(* CODESYS project 117_1_V0.5.project

Project tree, tasks and I/O mapping:
  Device : XSLH-30A32, Wuxi Xinje Electric Co.,Ltd., version 3.5.15.40_2.2.0_2023.07.04
      unmapped channels: IN, OUT
    application Application
      libraries: Standard, * (System); Util, * (System); CmpIecTask, 3.5.21.0 (System); Time and Date, 3.5.17.0 (3S - Smart Software Solutions GmbH); Asynchronous Job  Manager, 3.5.19.0 (3S - Smart Software Solutions GmbH); CmpEventMgr, 3.5.14.0 (System); Component Manager, 3.5.13.0 (System); CmpApp, 3.5.15.0 (System)
      task EtherCAT_Task (cyclic, interval 4 ms, priority 1) calls nothing
      task MainTask (cyclic, interval 4 ms, priority 8) calls MAIN
      6.Logic/
        data type STATUS
        function block StandLogic [ST]: _move_algorythm, _get_status, _change_control_mode, _jogging, _init, _alarm_notification, _read_inputs, _collect_errors, _driver_power, _write_outputs, _reset_alarms, _check_exciter, read_control_mode, _check_removing_limit_switch
        data type AUTO_MOVE_STEPS
        data type CONTROL_MODE
      Symbols
      0.TaskData/
        TimeManager_Structs/
          data type MEASUREMENT_UNITS
          data type TYPE_
        function block TimeManager [ST]: get_date_time, get_interval_time_type_INT, get_interval_time_type_REAL, get_interval_time_type_TIME, get_interval_time_type_UINT, get_cycle_count
      1.IO/
        Output/
          function block OutputManager [ST]: set_data
          data type DQ_VARS
        Input/
          function block InputManager [ST]: get_analog_data, get_discrete_data
          data type ALL_DI
          data type ALL_AI
      2.PID/
        PID_Structs/
          data type PID_STATUS_UDT
          data type PID_DIRECTION_UDT
          data type PID_DIAGNOSTIC_UDT
          data type PID_PARAMETERS_UDT
        function block BasicPIDController [ST]: Set_Configuration, Get_Diagnostics, xDifferential, Enable, Disable, xSp, xError, xPv, xIntegral, xOutput, Reset, xProportional
      2.Exciter/
        SwitchingAndFeedbackControl/
          data type SW_STATUS
          function block SwitchingWithFeedbackControl [ST]
          function block WaitingTimer [ST]
      4.Servo/
        Servo_Structs/
          data type ERROR_INDEX
          data type SMC_ERROR_TO_STRING
        function block SM3ServoDriver [ST]: _error_handler, set_power_on, stop_follow_velocity, start_forward_jogging, get_power_status, set_power_off, stop_jogging, reset_errors, start_follow_velocity, get_axis_errors, start_backward_jogging, get_axis_communication
      5.PRG/
        program MAIN [ST]
    Modbus_TCP : Modbus TCP, Wuxi Xinje Electric Co.,Ltd., version 3.0.0.0
    SoftMotion General Axis Pool
    EtherCAT_Master_SoftMotion : EtherCAT Master SoftMotion, CODESYS, version 4.10.0.0
        settings: SlaveAutoRestart = True; NetworkName = 'eth1'; NetworkName = "eth1"; SrcAddress1 = 26855; SrcAddress2 = 1253576340; EnableSecondAdapter = False
      ECAT_2057P_16DO : ECAT-2057P(RevC.) 16 K. Dig. Aus. Source 40V 0.3A, ICP DAS Co., Ltd., order no. ECAT-2057P 16DO, version Revision=16#00400001
          settings: Physical Address of the Slave = 1002; AutoIncr Address of the Slave = 4294967295; StationAlias = 0; FMMU.Global Start Address = 16#02000000; FMMU.Physical Start Address = 16#0F00; FMMU.Access = 16#02; DC sync0 cycletime = 4000; DC sync1 cycletime = 4000
          unmapped channels: Output 0 to 7, Output 0 to 7, Output 0 to 7, Output 0 to 7, Output 0 to 7, Output 0 to 7, Output 0 to 7, Output 0 to 7, Output 8 to 15, Output 8 to 15, Output 8 to 15, Output 8 to 15, Output 8 to 15, Output 8 to 15, Output 8 to 15, Output 8 to 15
      SD700_ECAT_Drive : SD700_ECAT_V1.5_G, Shenzhen Veichi Electric Co., Ltd, order no. SD700_ECAT Drive, version Revision=16#02040608
          settings: Number of Inputs = 7; Number of Infos about Inputs = 7; EnableExpertSettings = True; Watchdog_Reg_0400 = 2498; Watchdog_Reg_0410 = 1000; Watchdog_Reg_0420 = 1000; Physical Address of the Slave = 1003; AutoIncr Address of the Slave = 4294967294; StationAlias = 0; Sync.Length = 18; FMMU.Global Start Address = 16#02000002; FMMU.Physical Start Address = 16#1100; FMMU.Access = 16#02; FMMU.Global Start Address = 16#01000002; FMMU.Length = 18; FMMU.Physical Start Address = 16#1400; FMMU.Access = 16#01; FMMU.Global Start Address = 16#00080000; FMMU.Physical Start Address = 16#080D; FMMU.Access = 16#01; DC sync0 cycletime = 4000; DC enable = 1; DC sync0 enable = 1; DC sync0 shift time = 0; DC sync1 cycletime = 4000; DC sync1 enable = 0; DC sync1 factor = 'x 1'; DC sync1 shift time = 0; Number of SDO = 3; Interpolation time period.Value = 4; RxTxPdo.NumberofEntries = 7; RxTxPdo.Index = 16#1A01; RxTxPdo.DependOnSlot = False; RxTxPdo.DependOnSlotGroup = False; RxTxPdo.OverwrittenByModule = False; Exclude = [16#1A00,16#1A02,16#1A03]; Status Word.Offset = 0; Status Word.DependOnSlot = False; Status Word.DependOnSlotGroup = False; ActualPosition.Offset = 0;
            ActualPosition.DependOnSlot = False; ActualPosition.DependOnSlotGroup = False; Velocity actual value.Offset = 0; Velocity actual value.DependOnSlot = False; Velocity actual value.DependOnSlotGroup = False; Un000.Index = 16#3000; Un000.SubIndex = 0; Un000.Size = 16; Un000.Offset = 0; Un000.DependOnSlot = False; Un000.DependOnSlotGroup = False; Un001.Index = 16#3001; Un001.SubIndex = 0; Un001.Size = 16; Un001.Offset = 0; Un001.DependOnSlot = False; Un001.DependOnSlotGroup = False; Un004.Index = 16#3004; Un004.SubIndex = 0; Un004.Size = 16; Un004.Offset = 0; Un004.DependOnSlot = False; Un004.DependOnSlotGroup = False; Un005.Index = 16#3005; Un005.SubIndex = 0; Un005.Size = 16; Un005.Offset = 0; Un005.DependOnSlot = False; Un005.DependOnSlotGroup = False; Status Word.Default = ''; Status Word.Comment = ''; ActualPosition.Default = ''; ActualPosition.Comment = ''; Velocity actual value.Default = ''; Velocity actual value.Comment = ''; Un000.Name = 'Un000'; Un000.DataType = 'INT'; Un000.Default = ''; Un000.Comment = ''; Un001.Name = 'Un001';
            Un001.DataType = 'INT'; Un001.Default = ''; Un001.Comment = ''; Un004.Name = 'Un004'; Un004.DataType = 'UINT'; Un004.Default = ''; Un004.Comment = ''; Un005.Name = 'Un005'; Un005.DataType = 'UINT'; Un005.Default = ''; Un005.Comment = ''
          unmapped channels: Control Word, TargetPosition, TargetVelocity, Status Word, ActualPosition, Velocity actual value, Un000, Un001, Un004, Un005
        SM_Drive_GenericDSP402 : SM_Drive_GenericDSP402, CODESYS, order no. 0, version 4.19.0.0
            settings: wDriveID = 0; dwRatioTechUnitsDenom = 83886080; eRampType = 0; ScalingIncs = 8388608; ScalingMotorTurns2 = 50; ScalingUnits = 5; AdrOffset_8010 = 4; BitOffset_8010 = 0; BitLength_8010 = 16; Address_8010 = '%QW2'; Type_8010 = 'UINT'; AddressPointer_8010 = ADR(%QW2); AdrOffset_8020 = 8; BitOffset_8020 = 0; BitLength_8020 = 32; Address_8020 = '%QD2'; Type_8020 = 'DINT'; AddressPointer_8020 = ADR(%QD2); AdrOffset_8030 = 12; BitOffset_8030 = 0; BitLength_8030 = 32; Address_8030 = '%QD3'; Type_8030 = 'DINT'; AddressPointer_8030 = ADR(%QD3); AdrOffset_8040 = 4294967295; BitOffset_8040 = 0; BitLength_8040 = 16; Address_8040 = ''; Type_8040 = 'INT'; AddressPointer_8040 = 0; AdrOffset_8050 = 4294967295; BitOffset_8050 = 0; BitLength_8050 = 8; Address_8050 = ''; Type_8050 = 'SINT'; AddressPointer_8050 = 0; AdrOffset_8060 = 4294967295; BitOffset_8060 = 0; BitLength_8060 = 16; Address_8060 = '';
              Type_8060 = 'UINT'; AddressPointer_8060 = 0; AdrOffset_8070 = 4294967295; BitOffset_8070 = 0; BitLength_8070 = 0; Address_8070 = ''; Type_8070 = ''; AddressPointer_8070 = 0; AdrOffset_8080 = 4294967295; BitOffset_8080 = 0; BitLength_8080 = 0; Address_8080 = ''; Type_8080 = ''; AddressPointer_8080 = 0; AdrOffset_8090 = 4294967295; BitOffset_8090 = 0; BitLength_8090 = 0; Address_8090 = ''; Type_8090 = ''; AddressPointer_8090 = 0; AdrOffset_8510 = 4; BitOffset_8510 = 0; BitLength_8510 = 16; Address_8510 = '%IW2'; Type_8510 = 'UINT'; AddressPointer_8510 = ADR(%IW2); AdrOffset_8520 = 8; BitOffset_8520 = 0; BitLength_8520 = 32; Address_8520 = '%ID2'; Type_8520 = 'DINT'; AddressPointer_8520 = ADR(%ID2); AdrOffset_8530 = 12; BitOffset_8530 = 0; BitLength_8530 = 32; Address_8530 = '%ID3'; Type_8530 = 'DINT'; AddressPointer_8530 = ADR(%ID3); AdrOffset_8540 = 4294967295; BitOffset_8540 = 0;
              BitLength_8540 = 16; Address_8540 = ''; Type_8540 = 'INT'; AddressPointer_8540 = 0; AdrOffset_8550 = 4294967295; BitOffset_8550 = 0; BitLength_8550 = 0; Address_8550 = ''; Type_8550 = ''; AddressPointer_8550 = 0; AdrOffset_8560 = 4294967295; BitOffset_8560 = 0; BitLength_8560 = 32; Address_8560 = ''; Type_8560 = 'UDINT'; AddressPointer_8560 = 0; AdrOffset_8570 = 4294967295; BitOffset_8570 = 0; BitLength_8570 = 16; Address_8570 = ''; Type_8570 = 'UINT'; AddressPointer_8570 = 0; AdrOffset_8580 = 4294967295; BitOffset_8580 = 0; BitLength_8580 = 32; Address_8580 = ''; Type_8580 = 'DINT'; AddressPointer_8580 = 0; AdrOffset_8590 = 4294967295; BitOffset_8590 = 0; BitLength_8590 = 0; Address_8590 = ''; Type_8590 = ''; AddressPointer_8590 = 0; AdrOffset_8600 = 4294967295; BitOffset_8600 = 0; BitLength_8600 = 0; Address_8600 = ''; Type_8600 = ''; AddressPointer_8600 = 0;
              AdrOffset_8600 = 4294967295; BitOffset_8600 = 0; BitLength_8600 = 0; Address_8610 = ''; Type_8610 = ''; AddressPointer_8610 = 0; AdrOffset_8620 = 4294967295; BitOffset_8620 = 0; BitLength_8620 = 0; Address_8620 = ''; Type_8620 = ''; AddressPointer_8620 = 0
      ECAT_2016N_1 : ECAT-2016N 1 K. Ana. Eingang, Diff., 16-bit, ICP DAS Co.LTD, order no. ECAT-2016N , version Revision=16#00100001
          settings: EnableExpertSettings = True; StationAlias = 0; DC sync0 cycletime = 4000; DC sync1 cycletime = 4000
          unmapped channels: Status__Underrange, Status__Overrange, Status__Limit 1, Status__Limit 1, Status__Limit 2, Status__Limit 2, Status__Error, ---, ---, ---, ---, ---, ---, ---, Status__TxPDO State, Status__TxPDO Toggle, Value
      ECAT_2053_16DI : ECAT-2053 16 K. Dig. Ein. Wet 50V, ICP DAS Co., Ltd., order no. ECAT-2053 16DI, version Revision=16#00000001
          settings: Physical Address of the Slave = 1001; StationAlias = 1001; Optional = False; DeviceIdenticationADO = 0; DeviceIdenticationMode = 0; FMMU.Global Start Address = 16#01000000; FMMU.Physical Start Address = 16#1000; FMMU.Access = 16#01; DC sync0 cycletime = 4000; DC sync1 cycletime = 4000
          unmapped channels: Input 0 to 7, Input 0 to 7, Input 0 to 7, Input 0 to 7, Input 0 to 7, Input 0 to 7, Input 0 to 7, Input 0 to 7, Input 8 to 15, Input 8 to 15, Input 8 to 15, Input 8 to 15, Input 8 to 15, Input 8 to 15, Input 8 to 15, Input 8 to 15
      ECAT_2016N : ECAT-2016N 1 K. Ana. Eingang, Diff., 16-bit, ICP DAS Co.LTD, order no. ECAT-2016N , version Revision=16#00100001
          settings: EnableExpertSettings = True; Physical Address of the Slave = 1004; AutoIncr Address of the Slave = 4294967293; StationAlias = 0; FMMU.Global Start Address = 16#0200000C; FMMU.Physical Start Address = 16#1100; FMMU.Access = 16#02; FMMU.Global Start Address = 16#01000014; FMMU.Physical Start Address = 16#1400; FMMU.Access = 16#01; FMMU.Global Start Address = 16#00080000; FMMU.StartBit = 1; FMMU.EndBit = 1; FMMU.Physical Start Address = 16#080D; FMMU.Access = 16#01; DC sync0 cycletime = 4000; DC enable = 0; DC sync0 enable = 0; DC sync0 shift time = 0; DC sync1 cycletime = 4000; DC sync1 enable = 0; DC sync1 shift time = 0; Number of SDO = 0
          unmapped channels: Status__Underrange, Status__Overrange, Status__Limit 1, Status__Limit 1, Status__Limit 2, Status__Limit 2, Status__Error, ---, ---, ---, ---, ---, ---, ---, Status__TxPDO State, Status__TxPDO Toggle, Value
      TEC_Sensor : TEC Sensor E101 mit 1 Magnet, ZDJY TEC Corp, order no. TEC Sensor, version Revision=16#000100C9
          settings: EnableExpertSettings = True; Physical Address of the Slave = 1005; AutoIncr Address of the Slave = 4294967292; StationAlias = 0; FMMU.Global Start Address = 16#01000018; FMMU.Physical Start Address = 16#1400; FMMU.Access = 16#01; DC sync0 cycletime = 4000; DC sync1 cycletime = 4000
          unmapped channels: Status 1, Position 1, Velocity 1
    Local High Speed IO
        unmapped channels: IN, OUT
  ГОСТ/
    data type E_I_II
    Р ИСО 15032-2001/
      data type E_A
      function block TestingForces_150321 [ST]
     Р53868-2021/
      data type E_P1_2
      function block TestingForces_53868 [ST]
    Р ИСО 10328-2021/
      function block TestingForces_10328 [ST]
      data type E_P3_8
*)

// Device/Application/4.Servo/Servo_Structs/ERROR_INDEX
TYPE ERROR_INDEX :
(
	communication,
	power,
	jogging,
	follow,
	reset,
	lastIndex
)UINT;
END_TYPE

// Device/Application/6.Logic/STATUS
{attribute 'strict'}
TYPE STATUS :
(
	NOT_COMMUNICATION,
	OFF,
	READY,
	MOVING,
	ERROR
);
END_TYPE

// ГОСТ/E_I_II
{attribute 'strict'}
TYPE E_I_II :
(
	I := 0,
	II := 1
);
END_TYPE

// Device/Application/2.Exciter/SwitchingAndFeedbackControl/SW_STATUS
{attribute 'qualified_only'}
{attribute 'strict'}
TYPE SW_STATUS :
(	
	NONE,
	WAITING,
	DONE,
	TIMEOUT_ERROR
);
END_TYPE

// ГОСТ/ Р53868-2021/E_P1_2
{attribute 'strict'}
TYPE E_P1_2 :
(
	P1:= 0,
	P2:= 1
);
END_TYPE

// ГОСТ/Р ИСО 15032-2001/E_A
{attribute 'strict'}
TYPE E_A :
(
	A60		:= 0,
	A80		:= 1,
	A100	:= 2
);
END_TYPE

// Device/Application/6.Logic/AUTO_MOVE_STEPS
{attribute 'strict'}
TYPE AUTO_MOVE_STEPS :
(
	AWAIT,
	INJECTION,
	RETENTION,
	FAILING
);
END_TYPE

// Device/Application/0.TaskData/TimeManager_Structs/MEASUREMENT_UNITS
{attribute 'strict'}
TYPE MEASUREMENT_UNITS  :
(
	MS,
	US
);
END_TYPE

// Device/Application/2.PID/PID_Structs/PID_STATUS_UDT
{attribute 'strict' := ''}
TYPE PID_STATUS_UDT :
(
	Disabled,
	Enabled
);
END_TYPE

// Device/Application/1.IO/Input/ALL_DI
{attribute 'strict'}
TYPE ALL_DI :
(
	inLiveCircuitsDC		,			
	inFirstAlarmMushroom	,
	inSecondAlarmMushroom	,
	inLiveCircuitsAC		,		
	inUpsDC_OK				,			
	inUpsBattaryBad			,		
	inUpsBattaryWork		,	
	inUpperLimitSwitch		,	
	inLowerLimitSwitch		,	
	inRemovingLimitSwitch	,
	inExciter				,		
	inBit11					,				
	inBit12					,				
	inLeftDoor				,			
	inRightDoor				,			
	inBit15					
);
END_TYPE

// Device/Application/2.PID/PID_Structs/PID_DIRECTION_UDT
{attribute 'strict' := ''}
TYPE PID_DIRECTION_UDT :
(
	///[0] Прямая работа: ошибка = SP - PV
	DIRECT,
	///[1] Обратная работа: ошибка = PV - SP
	REVERSE
);
END_TYPE

// Device/Application/6.Logic/CONTROL_MODE
{attribute 'strict'}
TYPE CONTROL_MODE :
(
	MANUAL	:= 10,
	AUTO	:= 20
);
END_TYPE

// Device/Application/2.PID/PID_Structs/PID_DIAGNOSTIC_UDT
TYPE PID_DIAGNOSTIC_UDT :
STRUCT
	Error			: REAL;
	PreviousError	: REAL;
	Proportional	: REAL;
	Integral		: REAL;
	Differential	: REAL;
	Status			: PID_STATUS_UDT;
	Direction		: PID_DIRECTION_UDT;
	Kp				: REAL;
	Ki				: REAL;
	Kd				: REAL;
	Ts				: TIME;
	MinOut			: REAL;
	MaxOut			: REAL;
END_STRUCT
END_TYPE

// ГОСТ/Р ИСО 10328-2021/E_P3_8
{attribute 'strict'}
TYPE E_P3_8 :
(
	P3:= 0,
	P4:= 1,
	P5:= 2,
	P6:= 3,
	P7:= 4,
	P8:= 5
	
);
END_TYPE

// Device/Application/2.PID/PID_Structs/PID_PARAMETERS_UDT
TYPE PID_PARAMETERS_UDT :
STRUCT
	Pv: REAL;
	Sp: REAL;
	Kp: REAL;
	Ki: REAL;
	Kd: REAL;
	Ts: TIME;
	MinOut: REAL;
	MaxOut: REAL;
	Direction: PID_DIRECTION_UDT;
END_STRUCT
END_TYPE

// Device/Application/1.IO/Input/ALL_AI
TYPE ALL_AI :
(
	tenza1000kgSensor,
	tenza50kgSensor	,
	motionSensor	,
    lastAnalogInIndex	
);
END_TYPE

// Device/Application/4.Servo/Servo_Structs/SMC_ERROR_TO_STRING
{attribute 'to_string'}
TYPE SMC_ERROR_TO_STRING :
(
	SMC_NO_ERROR := 0,
	SMC_DI_GENERAL_COMMUNICATION_ERROR := 1,
	SMC_DI_AXIS_ERROR := 2,
	SMC_DI_FIELDBUS_LOST_SYNCRONICITY := 3,
	SMC_DI_SWLIMITS_EXCEEDED := 10,
	SMC_DI_HWLIMITS_EXCEEDED := 11,
	SMC_DI_LINEAR_AXIS_OUTOFRANGE := 12,
	SMC_DI_HALT_OR_QUICKSTOP_NOT_SUPPORTED := 13,
	SMC_DI_VOLTAGE_DISABLED := 14,
	SMC_DI_IRREGULAR_ACTPOSITION := 15,
	SMC_DI_POSITIONLAGERROR := 16,
	SMC_DI_HOMING_ERROR := 17,
	SMC_DI_LICENSING_ERROR := 18,
	SMC_DI_DRIVE_LIMIT_ACTIVE := 19,
	SMC_REGULATOR_OR_START_NOT_SET := 20,
	SMC_WRONG_CONTROLLER_MODE := 21,
	SMC_INVALID_ACTION_FOR_LOGICAL := 25,
	SMC_AXIS_IS_NOT_OPERATIONAL := 27,
	SMC_AXIS_NOT_FOLLOWING_SETVALUES := 28,
	SMC_FB_WASNT_CALLED_DURING_MOTION := 30,
	SMC_AXIS_IS_NO_AXIS_REF := 31,
	SMC_AXIS_REF_CHANGED_DURING_OPERATION := 32,
	SMC_FB_ACTIVE_AXIS_DISABLED := 33,
	SMC_AXIS_NOT_READY_FOR_MOTION := 34,
	SMC_AXIS_ERROR_DURING_MOTION := 35,
	SMC_FB_CALLED_FROM_WRONG_TASK := 36,
	SMC_INVALID_DISTRIBUTED_CLOCKS_SETTINGS := 37,
	SMC_INVALID_TIMESTAMP := 38,
	SMC_AXIS_ERROR_DUE_TO_FB_ERROR := 39,
	SMC_VD_MAX_VELOCITY_EXCEEDED := 40,
	SMC_VD_MAX_ACCELERATION_EXCEEDED := 41,
	SMC_VD_MAX_DECELERATION_EXCEEDED := 42,
	SMC_3SH_INVALID_VELACC_VALUES := 50,
	SMC_3SH_MODE_NEEDS_HWLIMIT := 51,
	SMC_FRC_NO_FREE_HANDLE := 60,
	SMC_MAC_INITIALIZATION_FAILED := 65,
	SMC_MAC_INVALID_TASK_HANDLE := 66,
	SMC_MAC_TOO_MANY_TASKS := 67,
	SMC_MAC_ATOMIC_ADD_FAILED := 68,
	SMC_SDO_INVALID_DATALENGTH := 69,
	SMC_SCM_NOT_SUPPORTED := 70,
	SMC_SCM_AXIS_IN_WRONG_STATE := 71,
	SMC_SCM_INTERRUPTED := 72,
	SMC_ST_WRONG_CONTROLLER_MODE := 75,
	SMC_RAG_ERROR_DURING_STARTUP := 80,
	SMC_RAG_ERROR_AXIS_NOT_INITIALIZED := 81,
	SMC_PP_WRONG_AXIS_TYPE := 85,
	SMC_PP_NUMBER_OF_ABSOLUTE_BITS_INVALID := 86,
	SMC_NEGATIVE_MODULO_PERIOD := 87,
	SMC_CGR_ZERO_VALUES := 90,
	SMC_CGR_DRIVE_POWERED := 91,
	SMC_CGR_INVALID_POSPERIOD := 92,
	SMC_CGR_POSPERIOD_NOT_INTEGRAL := 93,
	SMC_FRACTION_TECH_UNITS_INVALID := 94,
	SMC_SCALING_PARAMETERS_NOT_POSITIVE := 95,
	SMC_SCALING_SETTINGS_TOO_LARGE := 96,
	SMC_MODULO_PERIOD_TOO_MANY_DIGITS := 97,
	SMC_P_FTASKCYCLE_EMPTY := 110,
	SMC_R_NO_ERROR_TO_RESET := 120,
	SMC_R_DRIVE_DOESNT_ANSWER := 121,
	SMC_R_ERROR_NOT_RESETTABLE := 122,
	SMC_R_DRIVE_DOESNT_ANSWER_IN_TIME := 123,
	SMC_R_CANNOT_RESET_COMMUNICATION_ERROR := 124,
	SMC_RP_PARAM_UNKNOWN := 130,
	SMC_RP_REQUESTING_ERROR := 131,
	SMC_RP_DRIVE_PARAMETER_NOT_MAPPED := 132,
	SMC_RP_PARAM_CONVERSION_ERROR := 133,
	SMC_WP_PARAM_INVALID := 140,
	SMC_WP_SENDING_ERROR := 141,
	SMC_WP_DRIVE_PARAMETER_NOT_MAPPED := 142,
	SMC_WP_PARAM_CONVERSION_ERROR := 143,
	SMC_H_AXIS_WASNT_STANDSTILL := 170,
	SMC_H_AXIS_DIDNT_START_HOMING := 171,
	SMC_H_AXIS_DIDNT_ANSWER := 172,
	SMC_H_ERROR_WHEN_STOPPING := 173,
	SMC_H_AXIS_IN_ERRORSTOP := 174,
	SMC_H_SET_OP_MODE_HOMING_FAILED := 175,
	SMC_H_CHECK_SET_OP_MODE_HOMING_FAILED := 176,
	SMC_H_PRE_HOMING_CHECKS_FAILED := 177,
	SMC_MS_UNKNOWN_STOPPING_ERROR := 180,
	SMC_MS_INVALID_ACCDEC_VALUES := 181,
	SMC_MS_DIRECTION_NOT_APPLICABLE := 182,
	SMC_MS_AXIS_IN_ERRORSTOP := 183,
	SMC_BLOCKING_MC_STOP_WASNT_CALLED := 184,
	SMC_MS_AXIS_ALREADY_STOPPING := 185,
	SMC_UNKNOWN_TASK_INTERVAL := 200,
	SMC_MA_INVALID_VELACC_VALUES := 201,
	SMC_MA_INVALID_DIRECTION := 202,
	SMC_MR_INVALID_VELACC_VALUES := 226,
	SMC_MR_INVALID_DIRECTION := 227,
	SMC_OVR_INVALID_OVERRIDE_FACTORS := 231,
	SMC_INVALID_AXIS_FORECAST := 235,
	SMC_AXIS_FORECAST_NOT_SUPPORTED := 236,
	SMC_MAD_INVALID_VELACC_VALUES := 251,
	SMC_MAD_INVALID_DIRECTION := 252,
	SMC_MSI_INVALID_VELACC_VALUES := 276,
	SMC_MSI_INVALID_DIRECTION := 277,
	SMC_MSI_INVALID_EXECUTION_ORDER := 278,
	SMC_LOGICAL_NO_REAL_AXIS := 300,
	SMC_MV_INVALID_ACCDEC_VALUES := 301,
	SMC_MV_DIRECTION_NOT_APPLICABLE := 302,
	SMC_PP_ARRAYSIZE := 325,
	SMC_PP_STEP0MS := 326,
	SMC_VP_ARRAYSIZE := 350,
	SMC_VP_STEP0MS := 351,
	SMC_AP_ARRAYSIZE := 375,
	SMC_AP_STEP0MS := 376,
	SMC_TP_TRIGGEROCCUPIED := 400,
	SMC_TP_COULDNT_SET_WINDOW := 401,
	SMC_TP_COMM_ERROR := 402,
	SMC_TRIGGER_OUT_OF_RANGE := 403,
	SMC_LATCH_IN_CONTROLLER_NOT_SUPPORTED := 404,
	SMC_AT_TRIGGERNOTOCCUPIED := 410,
	SMC_MCR_INVALID_VELACC_VALUES := 426,
	SMC_MCR_INVALID_DIRECTION := 427,
	SMC_MCA_INVALID_VELACC_VALUES := 451,
	SMC_MCA_INVALID_DIRECTION := 452,
	SMC_MCA_DIRECTION_NOT_APPLICABLE := 453,
	SMC_SDL_INVALID_AXIS_STATE := 475,
	SMC_SDL_INVALID_VELACC_VALUES := 476,
	SMC_SACF_INVALID_DYNAMIC_FACTOR := 480,
	SMC_INVALID_VELACCJERK_VALUES := 501,
	SMC_INVALID_DIRECTION := 502,
	SMC_CR_NO_TAPPETS_IN_CAM := 600,
	SMC_CR_TOO_MANY_TAPPETS := 601,
	SMC_CR_MORE_THAN_32_ACCESSES := 602,
	SMC_CI_NO_CAM_SELECTED := 625,
	SMC_CI_MASTER_OUT_OF_SCALE := 626,
	SMC_CI_RAMPIN_NEEDS_VELACC_VALUES := 627,
	SMC_CI_SCALING_INCORRECT := 628,
	SMC_CI_TOO_MANY_TAPPETS_PER_CYCLE := 629,
	SMC_CI_MORE_THAN_32_ACCESSES := 630,
	SMC_CI_MASTER_SYNC_POSITION_OUT_OF_SCALE := 631,
	SMC_CI_AVOID_REVERSAL_FOR_FINITE_AXIS := 632,
	SMC_CI_MASTERSTARTDISTANCE_MUST_BE_ZERO_BUFFERED := 633,
	SMC_CI_CAM_CHANGED_DURING_RAMP_IN_DIST := 634,
	SMC_CB_NOT_IMPLEMENTED := 640,
	SMC_GI_RATIO_DENOM := 675,
	SMC_GI_INVALID_ACC := 676,
	SMC_GI_INVALID_DEC := 677,
	SMC_GI_MASTER_REGULATOR_CHANGED := 678,
	SMC_GI_INVALID_JERK := 679,
	SMC_PH_INVALID_VELACCDEC := 725,
	SMC_PH_ROTARYAXIS_PERIOD0 := 726,
	SMC_MASTER_REGULATOR_CHANGED := 727,
	SMC_NO_CAM_REF_TYPE := 750,
	SMC_CAM_TABLE_DOES_NOT_COVER_MASTER_SCALE := 751,
	SMC_CAM_TABLE_EMPTY_MASTER_RANGE := 752,
	SMC_CAM_TABLE_INVALID_MASTER_MINMAX := 753,
	SMC_CAM_TABLE_INVALID_SLAVE_MINMAX := 754,
	SMC_CAM_INVALID_ELEMENT_COUNT := 755,
	SMC_CAM_UNKNOWN_SEGMENT_TYPE := 756,
	SMC_SAFE_CAM_REF_ONLY_ONE_ACCESS_ALLOWED_AT_A_TIME := 757,
	SMC_CAM_REF_INSUFFICIENT_MEMORY := 758,
	SMC_GIP_MASTER_DIRECTION_CHANGE := 775,
	SMC_GIP_SLAVE_REVERSAL_CANNOT_BE_AVOIDED := 776,
	SMC_GIP_AVOID_REVERSAL_FOR_FINITE_AXIS := 777,
	SMC_GIP_MASTERSTARTDISTANCE_MUST_BE_ZERO_BUFFERED := 778,
	SMC_GIP_CANNOT_START_SYNC := 779,
	SMC_RAMP_IN_MASTER_DIRECTION_CHANGED := 780,
	SMC_RAMP_IN_SLAVE_REVERSAL_CANNOT_BE_AVOIDED := 781,
	SMC_DCS_ON_OFF_COMPENSATION_REQUIRES_FORECAST := 790,
	SMC_DCS_ON_OFF_COMPENSATION_EXCEEDS_FORECAST := 791,
	SMC_DCS_SWITCHES_MUST_BE_ORDERED_BY_POSITION := 792,
	SMC_DCS_SWITCHES_MUST_NOT_OVERLAP := 793,
	SMC_DCS_INVALID_TRACK_NUMBER := 794,
	SMC_DCS_MAX_SWITCHES_PER_TRACK_EXCEEDED := 795,
	SMC_DCS_SWITCH_POSITION_OUTSIDE_MODULO_PERIOD := 796,
	SMC_DCS_CAM_SWITCH_POINTER_NOT_SET := 797,
	SMC_BC_BL_TOO_BIG := 800,
	SMC_QPROF_DIVERGES := 825,
	SMC_QPROF_INVALID_PARAMETER := 826,
	SMC_QPROF_NO_RESULT := 827,
	SMC_QPROF_INVALID_NEW_LBD := 828,
	SMC_QPROF_BAD_NEGOTIATION := 829,
	SMC_QPROF_INVALID_INTERVAL := 830,
	SMC_QPROF_NOT_ENOUGH_PHASES := 831,
	SMC_TG_INTERNAL_ERROR := 832,
	SMC_SRT_NOT_STANDSTILL_OR_POWEROFF := 850,
	SMC_SRT_INVALID_RAMPTYPE := 851,
	SMC_SMT_NOT_STANDSTILL_OR_POWEROFF := 852,
	SMC_SMT_INVALID_MOVEMENTTYPE_OR_POSITIONPERIOD := 853,
	SMC_SMT_AXIS_NOT_VIRTUAL := 854,
	SMC_NO_LICENSE := 1000,
	SMC_INT_VEL_ZERO := 1001,
	SMC_INT_NO_STOP_AT_END := 1002,
	SMC_INT_DATA_UNDERRUN := 1003,
	SMC_INT_VEL_NONZERO_AT_STOP := 1004,
	SMC_INT_TOO_MANY_RECURSIONS := 1005,
	SMC_INT_NO_CHECKVELOCITIES := 1006,
	SMC_INT_PATH_EXCEEDED := 1007,
	SMC_INT_VEL_ACC_DEC_ZERO := 1008,
	SMC_INT_DWIPOTIME_ZERO := 1009,
	SMC_INT_JERK_NONPOSITIVE := 1010,
	SMC_INT_QPROF_DIVERGES := 1011,
	SMC_INT_INVLALID_VELOCITY_MODE := 1012,
	SMC_INT_TOO_MANY_AXES_INTERPOLATED := 1013,
	SMC_INT_DEGENERATE_SEGMENT := 1014,
	SMC_HIGH_CURVATURE_SPLINE := 1015,
	SMC_INT_PROBE_ACKNOWLEDGED_WHILE_MOVING := 1016,
	SMC_INT_PROBE_NOT_ACKNOWLEDGED := 1017,
	SMC_INT_PROBE_INTERNAL_ERROR := 1018,
	SMC_INT2DIR_BUFFER_TOO_SMALL := 1050,
	SMC_INT2DIR_PATH_FITS_NOT_IN_QUEUE := 1051,
	SMC_XINT_INVALID_DIRECTION := 1070,
	SMC_XINT_NOINTERSECTION := 1071,
	SMC_WAR_INT_OUTQUEUE_TOO_SMALL := 1080,
	SMC_WAR_END_VELOCITIES_INCORRECT := 1081,
	SMC_CV_ACC_DEC_VEL_NONPOSITIVE := 1100,
	SMC_CA_INVALID_ACCDEC_VALUES := 1120,
	SMC_TOK_INCOMPLETE_TOKEN_AT_END_OF_INPUT := 1130,
	SMC_TOK_NOT_A_VALID_TOKEN := 1131,
	SMC_TOK_AMBIGUOUS_INPUT := 1132,
	SMC_TOK_STRING_TOO_LONG_FOR_TOKEN := 1133,
	SMC_TOK_INVALID_NUMLIT := 1134,
	SMC_PRS_FUNC_DECL_TOO_FEW_ARGUMENTS := 1150,
	SMC_PRS_FUNC_DECL_TOO_MANY_ARGUMENTS := 1151,
	SMC_PRS_FUNC_DECL_WRONG_ARGUMENT_TYPE := 1152,
	SMC_PRS_LOCAL_VAR_NOT_FOUND := 1153,
	SMC_PRS_INVALID_STRING := 1154,
	SMC_PRS_TOO_MANY_CLOSING_BRACKETS := 1155,
	SMC_PRS_TOO_MANY_OPENING_BRACKETS := 1156,
	SMC_PRS_NO_SUCH_INFIX_OPERATOR := 1157,
	SMC_PRS_NO_SUCH_PREFIX_OPERATOR := 1158,
	SMC_PRS_OPERATOR_INVALID_PRECEDENCE := 1159,
	SMC_PRS_NOT_A_TERM := 1160,
	SMC_PRS_EXPRESSION_INVALID_SEQUENCE := 1161,
	SMC_PRS_TOO_MANY_TERMS := 1162,
	SMC_PRS_STACK_OVERFLOW := 1163,
	SMC_PRS_VAR_NAME_ALREADY_USED := 1164,
	SMC_PRS_INCOMPLETE_SENTENCE_IN_TOKEN_QUEUE := 1165,
	SMC_PRS_TOO_MANY_SUBPROGRAMS := 1167,
	SMC_PRS_TOO_MANY_SUBPROGRAM_PARAMETERS := 1168,
	SMC_PRS_SUBPROGRAM_LOOKUP_FAILED := 1169,
	SMC_PRS_VAR_NOT_FOUND := 1170,
	SMC_PRS_TOKEN_TYPE_UNKNOWN := 1171,
	SMC_PRS_GOT_NO_TERM := 1172,
	SMC_PRS_INVALID_VAR_TYPE := 1173,
	SMC_PRS_UNEXPECTED_TOKEN := 1174,
	SMC_PRS_ID3_EXPECTED := 1175,
	SMC_PRS_ID_TOO_LONG := 1176,
	SMC_PRS_GADDRESS_EXPECTED := 1177,
	SMC_PRS_NWORD_EXPECTED := 1178,
	SMC_PRS_NWORD_INVALID_SENTENCE_NUMBER := 1179,
	SMC_PRS_NWORD_SENTENCE_NUMBER_NO_NUMBER_LITERAL := 1180,
	SMC_PRS_USE_OF_RESERVED_KEYWORD := 1181,
	SMC_PRS_SUBPROGRAMS_SIGNATURE_MISMATCH := 1182,
	SMC_PRS_INITIAL_VALUE_HAS_WRONG_TYPE := 1183,
	SMC_PRS_TOO_MANY_LOCAL_VARIABLES := 1184,
	SMC_PRS_SUBPROG_MUST_BE_FIRST_SENTENCE := 1185,
	SMC_PRS_ONLY_ONE_SUBPROGRAM_PER_FILE_ALLOWED := 1186,
	SMC_PRS_LET_AFTER_REGULAR_SENTENCE := 1187,
	SMC_PRS_UNMATCHED_END_SUBPROGRAM := 1188,
	SMC_PRS_UNEXPECTED_TOKENS_AFTER_SUBPROGRAM := 1189,
	SMC_PRS_MISSING_END_SUBPROGRAM := 1190,
	SMC_PRS_USE_OF_KEYWORD := 1191,
	SMC_PRS_DYNCALL_EXPECTED_SUBNAME_EXP := 1192,
	SMC_PRS_DYNCALL_EXPECTED_SUBNAME_TYPE_STRING := 1193,
	SMC_DEC_ACC_TOO_LITTLE := 1200,
	SMC_DEC_RET_TOO_LITTLE := 1201,
	SMC_DEC_OUTQUEUE_RAN_EMPTY := 1202,
	SMC_DEC_JUMP_TO_UNKNOWN_LINE := 1203,
	SMC_DEC_INVALID_SYNTAX := 1204,
	SMC_DEC_3DMODE_OBJECT_NOT_SUPPORTED := 1205,
	SMC_DEC_NEGATIVE_PERIOD := 1206,
	SMC_DEC_DIMENSIONS_EXCLUSIVE_AU := 1207,
	SMC_DEC_DIMENSIONS_EXCLUSIVE_BV := 1208,
	SMC_DEC_DIMENSIONS_EXCLUSIVE_CW := 1209,
	SMC_DEC_DCS_NOT_ALL_OF_ABC_GIVEN := 1210,
	SMC_DEC_DCS_2D_NOT_IN_XY_PLANE := 1211,
	SMC_DEC_CIRCLE_NON_UNIFORM_SCALING := 1212,
	SMC_DEC_ROTATION_AFFECTS_SCALING := 1213,
	SMC_DEC_DCS_NOT_ALL_OF_IJK_GIVEN := 1214,
	SMC_IPR_LOCAL_VAR_UNKNOWN_TYPE := 1250,
	SMC_IPR_LVALUE_WRONG_TYPE := 1251,
	SMC_IPR_EVAL_STACK_OVERFLOW := 1252,
	SMC_IPR_NOT_A_NUMBER := 1253,
	SMC_IPR_DIVISION_BY_ZERO := 1254,
	SMC_IPR_INVALID_SCALING_FACTORS := 1255,
	SMC_IPR_INTERPRETER_STACK_IMBALANCE := 1256,
	SMC_IPR_INTERPRETER_STACK_OVERFLOW := 1257,
	SMC_IPR_INVALID_INTERPRETER_STACK_BUFFER := 1258,
	SMC_IPR_BUFFER_TOO_SMALL := 1259,
	SMC_NO_PROBE_ALLOWED := 1260,
	SMC_AT_MOST_ONE_PROBE_ALLOWED := 1261,
	SMC_PROBE_NON_POSITIVE := 1262,
	SMC_PROBE_TOO_LARGE := 1263,
	SMC_NO_HFUN_ON_PROBE_ALLOWED := 1264,
	SMC_ARC_2DMODE_K_AND_T_DETERMINE_APEX := 1265,
	SMC_ARC_RADIUS_AND_APEX_OR_CENTER_GIVEN := 1266,
	SMC_ARC_CENTER_NOT_GIVEN := 1267,
	SMC_ARC_DISTANCE_LARGER_THAN_DIAMETER := 1268,
	SMC_ARC_DISTANCE_TOO_SMALL := 1269,
	SMC_ARC_APEX_TOO_SMALL := 1270,
	SMC_ARC_APEX_TOO_LARGE := 1271,
	SMC_ARC_CENTER_NOT_ON_PERPENDICULAR_BISECTOR := 1272,
	SMC_CNC_INVALID_TWO_LETTER_TOKEN := 1273,
	SMC_CNC_ONLY_ONE_G_OR_M_WORD_ALLOWED := 1274,
	SMC_DEC_UNKNOWN_GWORD := 1275,
	SMC_CNC_POS_VALUES_NOT_SUPPORTED := 1276,
	SMC_CNC_SPLINE_ABORTED_BY_G75 := 1277,
	SMC_DNCCS_NO_DATA := 1280,
	SMC_DNCCS_TOO_MANY_CALLSTACKS := 1281,
	SMC_DNCCS_INVALID_PROGRAM_INDEX := 1282,
	SMC_DNCCS_TOO_MANY_PROGRAMS := 1283,
	SMC_DNCCS_WRONG_TASK := 1284,
	SMC_GCV_BUFFER_TOO_SMALL := 1300,
	SMC_GCV_BUFFER_WRONG_TYPE := 1301,
	SMC_GCV_UNKNOWN_IPO_LINE := 1302,
	SMC_CNC_INTERNAL_ERROR := 1400,
	SMC_PATH_MAX_HPOINTS_EXCEEDED := 1401,
	SMC_TRC_G75_NOT_ALLOWED := 1410,
	SMC_TRC_QUEUE_FULL_NON_CARTESIAN := 1411,
	SMC_TRC_SPLINE3D_5_NOT_SUPPORTED := 1412,
	SMC_TRC_ELLIPSES_NOT_SUPPORTED := 1413,
	SMC_TRC_PLANE_CHANGE_NOT_ALLOWED := 1414,
	SMC_CNC_INVALID_GEOINFO := 1415,
	SMC_CNC_CANNOT_APPEND_TO_OUTQUEUE := 1416,
	SMC_CNC_APPEND_ON_FIRST_RISING_EDGE := 1417,
	SMC_PROBE_G31_NOT_ALLOWED := 1418,
	SMC_AL_ELLIPSES_NOT_SUPPORTED := 1430,
	SMC_NAV_MAX_SUBPROGRAM_NESTING_EXCEEDED := 1450,
	SMC_NAV_RETURN_FROM_MAIN := 1451,
	SMC_NAV_SUBPROGRAM_DECLARATION_NOT_FOUND := 1452,
	SMC_NAV_NOT_ENOUGH_SPACE_FOR_COMPLETE_SENTENCE := 1453,
	SMC_NO_CNC_REF_TYPE := 1500,
	SMC_NO_OUTQUEUE_TYPE := 1501,
	SMC_GEOINFO_BUFFER_MISALIGNED := 1502,
	SMC_3D_MODE_NOT_SUPPORTED := 1600,
	SMC_SAA_SMOOTHAREA_TOO_LARGE := 1700,
	SMC_SAA_SP_INVALID_INPUT := 1701,
	SMC_SA_QUEUE_NOT_IN_BUFFER := 1800,
	SMC_SA_QUEUE_CHANGED_DURING_OP := 1801,
	SMC_OS_INVALID_PARAMETER := 1820,
	SMC_BSSP_IPO_NOT_ACTIVE := 1830,
	SMC_BS_SAVEDPOS_NOT_REACHED := 1831,
	SMC_BS_NO_POS_STORED := 1832,
	SMC_INVALID_FEATURE_FLAG := 1900,
	SMC_SMB_HFUN_NOT_SUPPORTED := 1901,
	SMC_SMB_ONLY_3DMODE := 1902,
	SMC_SMB_ERROR_COMPUTING_SPLINE := 1903,
	SMC_SMM_INVALID_PARAM_NUMBER := 1910,
	SMC_ORIENTATION_UNKNOWN := 1911,
	SMC_NOT_IMPLEMENTED := 1949,
	SMC_INVALID_PARAMETER := 1950,
	SMC_BLENDING_NOT_SUPPORTED_BY_PREVIOUS_MOVEMENT := 1951,
	SMC_BUFFERED_NOT_SUPPORTED_BY_PREVIOUS_MOVEMENT := 1952,
	SMC_INHERIT_OWNER_ACTIVE_MOVEMENT_NOT_CALLED := 1953,
	SMC_MOVING_WITHOUT_ACTIVE_MOVEMENT := 1954,
	SMC_BUFFER_MODE_NOT_SUPPORTED := 1955,
	SMC_ERROR_IN_A_PREVIOUS_MOVEMENT := 1956,
	SMC_MORE_THAN_ONE_MOVEMENT_PER_INSTANCE := 1957,
	SMC_SUPERIMPOSED_FB_WASNT_CALLED := 1958,
	SMC_RNCF_FILE_DOESNT_EXIST := 2000,
	SMC_RNCF_NO_BUFFER := 2001,
	SMC_RNCF_BUFFER_TOO_SMALL := 2002,
	SMC_RNCF_DATA_UNDERRUN := 2003,
	SMC_RNCF_VAR_COULDNT_BE_REPLACED := 2004,
	SMC_RNCF_NOT_VARLIST := 2005,
	SMC_RNCF_NO_STRINGBUFFER := 2006,
	SMC_RNCF_STRINGBUFFER_OVERRUN := 2007,
	SMC_RNCF_SUBPROGRAM_FILE_NOT_FOUND := 2008,
	SMC_RNCF_FILE_CANNOT_DETERMINE_SIZE := 2009,
	SMC_RNCQ_FILE_DOESNT_EXIST := 2050,
	SMC_RNCQ_NO_BUFFER := 2051,
	SMC_RNCQ_BUFFER_TOO_SMALL := 2052,
	SMC_RNCQ_UNEXPECTED_EOF := 2053,
	SMC_ADL_FILE_CANNOT_BE_OPENED := 2100,
	SMC_ADL_BUFFER_OVERRUN := 2101,
	SMC_RCAM_FILE_DOESNT_EXIST := 2200,
	SMC_RCAM_TOO_MUCH_DATA := 2201,
	SMC_RCAM_WRONG_COMPILE_TYPE := 2202,
	SMC_RCAM_WRONG_VERSION := 2203,
	SMC_RCAM_UNEXPECTED_EOF := 2204,
	SMC_RCAM_WRITE_ERROR := 2205,
	SMC_RCAM_READ_ERROR := 2206,
	SMC_WDPF_CHANNEL_OCCUPIED := 3001,
	SMC_WDPF_CANNOT_CREATE_FILE := 3002,
	SMC_WDPF_ERROR_WHEN_READING_PARAMS := 3003,
	SMC_WDPF_TIMEOUT_PREPARING_LIST := 3004,
	SMC_ENC_DENOM_ZERO := 5000,
	SMC_ENC_AXISUSEDBYOTHERFB := 5001,
	SMC_ENC_FILTER_DEPTH_INVALID := 5002,
	SMC_INTERNAL_ERROR_INIT_MOVEMENT := 6000,
	SMC_INVALID_AXIS_TYPE := 6001,
	SMC_PCCQ_POINTBUFFERTOOSMALL := 10000,
	SMC_PCCQ_INPUTBUFFERFULLBUTNOTFINALIZED := 10001,
	SMC_PCCQ_PATH_NOT_COMPLETELY_IN_INPUT_BUFFER := 10002,
	SMC_AXIS_GROUP_WRONG_STATE := 11000,
	SMC_AXIS_GROUP_TOO_MANY_AXES := 11001,
	SMC_AXIS_GROUP_INVALID_DYNLIMITS := 11002,
	SMC_AXIS_GROUP_INVALID_COORD_SYSTEM := 11004,
	SMC_AXIS_GROUP_SINGLE_AXIS_ERROR := 11005,
	SMC_MOVE_INVALID_BUFFER_MODE := 11006,
	SMC_MOVE_INVALID_DYNAMIC_FACTOR := 11007,
	SMC_MOVE_INVALID_DYNAMICS := 11008,
	SMC_AXIS_GROUP_AXIS_NOT_PART_OF_GROUP := 11009,
	SMC_AXIS_GROUP_NOT_SUPPORTED := 11010,
	SMC_AXIS_GROUP_KINEMATICS_NOT_SET := 11011,
	SMC_AXIS_GROUP_WRONG_NUMBER_OF_AXES := 11012,
	SMC_AXIS_GROUP_INTERRUPTED_BY_SINGLE_AXIS := 11013,
	SMC_AXIS_GROUP_FOLLOW_SETVALUES := 11014,
	SMC_AXIS_GROUP_TOO_MANY_DEPENDENCIES := 11015,
	SMC_AXIS_GROUP_MUTUAL_DEPENDENCY := 11016,
	SMC_AXIS_GROUP_DEPENDENCY_IN_DIFFERENT_TASK := 11017,
	SMC_AXIS_GROUP_AXIS_IN_DIFFERENT_TASK := 11018,
	SMC_AXIS_GROUP_PCS_STILL_IN_USE := 11019,
	SMC_AXIS_GROUP_CMD_ABORTED_DUE_TO_ERROR := 11020,
	SMC_AXIS_GROUP_INVALID_PARAMETER := 11021,
	SMC_AXIS_GROUP_UNSUPPORTED_RAMPTYPE := 11022,
	SMC_MOVE_INVALID_TRANSITION_PARAMETER := 11023,
	SMC_AXIS_GROUP_CPTR_CANNOT_FOLLOW := 11025,
	SMC_AXIS_GROUP_CONTINUE_WRONG_POSITION := 11026,
	SMC_AXIS_GROUP_CONTINUE_BUFFER_TOO_SMALL := 11027,
	SMC_AXIS_GROUP_CONTINUE_WRONG_CHECKSUM := 11028,
	SMC_AXIS_GROUP_IDLE_WAIT_AXES_MOVING := 11029,
	SMC_AXIS_INVERSE_TRAFO_EXCEEDING_POSLIMITS := 11030,
	SMC_AXIS_GROUP_CANNOT_ADD_SAME_AXIS := 11031,
	SMC_AXIS_GROUP_TRANSFORMATION_NOT_SET := 11032,
	SMC_AXIS_GROUP_NON_RESUMABLE_ERROR := 11033,
	SMC_AXIS_GROUP_CONTINUE_DATA_NOT_WRITTEN := 11034,
	SMC_AXIS_GROUP_INVALID_INTERRUPT_POSITION := 11036,
	SMC_RELATIVE_MOVEMENT_TRACKING_CS := 11037,
	SMC_RELATIVE_MOVEMENT_ABORTING_TRACKING := 11038,
	SMC_CIRCULAR_MOVEMENT_TRACKING_CS := 11039,
	SMC_CIRCULAR_MOVEMENT_ABORTING_TRACKING_CS := 11040,
	SMC_AXIS_GROUP_CONTINUE_POSITION_WRONG_CHECKSUM := 11041,
	SMC_CIRCULAR_TRACKING_TOOL_CHANGE_NOT_SUPPORTED := 11042,
	SMC_AXIS_GROUP_COULD_NOT_WRITE_CONTINUE_DATA := 11043,
	SMC_MODULO_AXIS_FOR_NON_ROTARY_JOINT := 11044,
	SMC_MODULO_AXIS_FOR_LIMITED_ROTARY_JOINT := 11045,
	SMC_MODULO_AXIS_PERIOD_NOT_360 := 11046,
	SMC_FB_WASNT_CALLED_DURING_EXECUTION := 11047,
	SMC_NO_EVALUATION_POSSIBLE_FOR_TIME_OFFSET := 11048,
	SMC_INVALID_SOURCE_TYPE_FOR_TIME_OFFSET := 11049,
	SMC_INVALID_TIME_OFFSET := 11050,
	SMC_TIME_OFFSET_TOO_LARGE := 11051,
	SMC_AXIS_GROUP_MAX_NUM_ADDITIONAL_AXES_EXCEEDED := 11052,
	SMC_INVALID_COORD_SYSTEM_FOR_TIME_OFFSET := 11053,
	SMC_KERNEL_PTP_INTERNAL_ERROR := 11100,
	SMC_KERNEL_PTP_INVALID_TASKCYCLETIME := 11101,
	SMC_TRAFO_INVALID_PARAMETERS := 12000,
	SMC_TRAFO_INVALID_CONSTELLATION := 12001,
	SMC_TRAFO_INVALID_COUPLING := 12002,
	SMC_TRAFO_NOT_INITIALIZED := 12003,
	SMC_TRAFO_NO_TOOL_WITH_OFFSET_ALLOWED := 12004,
	SMC_AXIS_GROUP_TOOL_OFFSET_INCOMPATIBLE_WITH_KINEMATICS := 12005,
	SMC_TRAFO_INVALID_AXIS_LIMITS := 12006,
	SMC_AXIS_GROUP_PATH_DEVIATION_TOO_HIGH := 12007,
	SMC_AXIS_POSITION_EXCEEDS_POSLIMITS := 12008,
	SMC_AXIS_GROUP_NO_DYNAMIC_MODEL_CONFIGURED := 12009,
	SMC_DYNAMICS_NUM_TORQUES_NEQ_NUM_AXES := 12010,
	SMC_AXIS_GROUP_MAX_AXIS_LAG_EXCEEDED := 12020,
	SMC_AXIS_GROUP_MAX_POSITION_LAG_EXCEEDED := 12021,
	SMC_AXIS_GROUP_MAX_ORIENTATION_LAG_EXCEEDED := 12022,
	SMC_CP_CACHE_FULL := 12100,
	SMC_CP_EVAL_ERROR := 12101,
	SMC_CP_NON_CONTINUABLE_STATE := 12102,
	SMC_CP_MAX_LENGTH_EXCEEDED := 12103,
	SMC_CP_ACCELERATION_TOO_HIGH := 12104,
	SMC_CP_MAX_ITERATIONS_EXCEEDED := 12105,
	SMC_CP_NO_TRAJECTORY := 12106,
	SMC_CP_OUT_QUEUE_FULL := 12107,
	SMC_CP_QUEUE_UNDERRUN := 12108,
	SMC_CP_INVALID_QUEUE := 12109,
	SMC_CP_BLENDING_INTERNAL_ERROR := 12110,
	SMC_CP_CIRCLE_COLLINEAR_POINTS := 12111,
	SMC_CP_CIRCLE_CENTER_NOT_ON_BISECTOR := 12112,
	SMC_CP_CIRCLE_RADIUS_ZERO := 12113,
	SMC_CP_CIRCLE_DISTANCE_LARGER_THAN_DIAMETER := 12114,
	SMC_CP_CIRCLE_START_AND_ENDPOINT_EQUAL := 12115,
	SMC_CP_BLENDING_DEGENERATE_SPLINE := 12116,
	SMC_CP_ELEMENT_TOO_SHORT := 12117,
	SMC_CP_COULD_NOT_CUT_PATH := 12118,
	SMC_CP_INVALID_ANGULAR_VEL_ACC := 12119,
	SMC_CP_INVALID_ORIENTATION := 12120,
	SMC_CP_TIME_BUDGET_EXCEEDED := 12121,
	SMC_AXIS_GROUP_AXIS_LIMIT_VIOLATED := 12122,
	SMC_CP_CONFIGS_DIFFER := 12125,
	SMC_CP_BUS_TASK_NOT_CALLED := 12126,
	SMC_CP_NO_ROOT_IN_INTERVAL_FOUND := 12127,
	SMC_CP_KIN_DOES_NOT_SUPPORT_AXIS_ORIENTATION_IPO := 12128,
	SMC_CP_AXIS_ORIENTATION_IPO_NOT_SUPPORTED_FOR_CPTR := 12129,
	SMC_CP_INVALID_PATH_ELEM := 12130,
	SMC_CP_TRANSITION_NOT_SMOOTH := 12131,
	SMC_CP_AXIS_ORIENTATION_IPO_CONFIG_DIFFERS := 12132,
	SMC_CP_AXIS_ORIENTATION_IPO_OFFSET2_NOT_IMPLEMENTED := 12133,
	SMC_CP_ROTARY_AXIS_PERIOD_MISMATCH := 12134,
	SMC_CP_ROTARY_AXIS_RANGE_VIOLATION := 12135,
	SMC_CP_COMPUTE_TARGET_DISCONTINUITY := 12136,
	SMC_CP_TRAJECTORY_NOT_SMOOTH := 12137,
	SMC_CP_ERROR_CREATING_PARAM_TRANSFORM := 12138,
	SMC_CP_PTP_DATA_NUMBER_OF_AXES := 12139,
	SMC_CP_NEGATIVE_PATH_VELOCITY := 12140,
	SMC_CP_TRANSITIONING_FROM_SINGLE_AXIS_MOVEMENT_NOT_SUPPORTED := 12141,
	SMC_CP_PLANNER_NO_PROGRESS := 12142,
	SMC_CP_INTERNAL_EVAL_CACHE_ERROR := 12143,
	SMC_CP_INVALID_ROOT_ACC_TOO_HIGH := 12144,
	SMC_CP_INVALID_ROOT_TRAJECTORY_TOO_LARGE := 12145,
	SMC_CP_EMPTY_TRAJECTORY := 12146,
	SMC_CP_FORECAST_TOO_LARGE := 12147,
	SMC_CP_INVALID_ROOT_ENDPOS_NOT_GREATER_STARTPOS := 12148,
	SMC_CP_AXIS_VELOCITY_LIMIT_EXCEEDED_WHITHOUT_MOVING := 12150,
	SMC_CP_AXIS_ACCELERATION_LIMIT_EXCEEDED_WHITHOUT_MOVING := 12151,
	SMC_CP_AXIS_JERK_LIMIT_EXCEEDED_WHITHOUT_MOVING := 12152,
	SMC_CP_AXIS_TORQUE_LIMIT_EXCEEDED_WHITHOUT_MOVING := 12153,
	SMC_GROUPJOG2_MAX_DISTANCE_NON_POSITIVE := 12200,
	SMC_GROUPJOG2_DYNAMIC_CS_NOT_SUPPORTED := 12201,
	SMC_TRIGGER_TOO_MANY_TRIGGERS_PREPARED := 12300,
	SMC_TRIGGER_UNSUPPORTED_MOVEMENT_TYPE := 12301,
	SMC_TRIGGER_INVALID_POS_TYPE := 12302,
	SMC_TRIGGER_RELATIVE_POSITION_OUT_OF_RANGE := 12303,
	SMC_TRIGGER_PLANE_NORMAL_NOT_A_UNIT := 12304,
	SMC_TRIGGER_PLANE_DISTANCE_NEGATIVE := 12305,
	SMC_TRIGGER_PLANE_COORD_SYSTEM_INVALID := 12306,
	SMC_TRIGGER_DISTANCE_OUT_OF_RANGE := 12307,
	SMC_TRIGGER_PLANE_NO_INTERSECTION := 12308,
	SMC_TRIGGER_TRACKING_TRANSITION_NOT_SUPPORTED := 12309,
	SMC_TRIGGER_PTP_NOT_SUPPORTED := 12310,
	SMC_CAM_BUILDER_FULL := 12400,
	SMC_CAM_BUILDER_INVALID_MASTER_DISTANCE := 12401,
	SMC_CAM_BUILDER_GAP_BETWEEN_SEGMENTS := 12402,
	SMC_CAM_BUILDER_NO_IMPLICIT_LEFT_BOUNDARY_ALLOWED := 12403,
	SMC_CAM_BUILDER_INVALID_IMPLICIT_CAM_SEGMENT_MASTER_DISTANCE := 12404,
	SMC_CAM_BUILDER_CAM_REF_INSUFFICIENT_MEMORY := 12405,
	SMC_CAM_BUILDER_LAST_SEGMENT_HAS_IMPLICIT_RIGHT_BOUNDARY := 12406,
	SMC_CAM_BUILDER_INVALID_CAM_REF_INITIALIZATION := 12407,
	SMC_CAM_BUILDER_ERROR_PENDING := 12408,
	SMC_CAM_BUILDER_CONTINUITY_REQUIREMENT_VIOLATED := 12409,
	SMC_CAM_BUILDER_MASTER_DISTANCE_TOO_SHORT := 12410,
	SMC_CAM_BUILDER_IMPLICIT_CAM_SEGMENT_DISTANCE_TOO_SHORT := 12411,
	SMC_CAM_BUILDER_CAM_REF_INVALID_ARRAY_SIZE := 12412,
	SMC_CAM_BUILDER_MODIFIED_SINE_INVALID_LAMBDA_OR_ACC_PARAM := 12415,
	SMC_CAM_BUILDER_MODIFIED_SINE_ACC_PARAM_RIGHT_BOUND_IMPLICIT := 12416,
	SMC_CAM_BUILDER_INVALID_COMPILE_TYPE := 12417,
	SMC_MOVEMENT_INTERNAL_ERROR := 13001,
	SMC_MOVEMENT_GET_POS_INTERNAL_ERROR := 13002,
	SMC_CPTR_INTERNAL_ERROR := 13003,
	SMC_CP_IPO_INTERNAL_ERROR := 13004,
	SMC_CP_ADD_NEW_MOVEMENT_INTERNAL_ERROR := 13005,
	SMC_AXIS_GROUP_COORDINATION_INTERNAL_ERROR := 13006,
	SMC_AXIS_GROUP_ADD_MOVEMENT_INTERNAL_ERROR := 13007,
	SMC_AXIS_GROUP_READ_AXIS_STATES_INTERNAL_ERROR := 13008,
	SMC_AXIS_GROUP_READ_VEL_INTERNAL_ERROR := 13009,
	SMC_AXIS_GROUP_READ_ACC_INTERNAL_ERROR := 13010,
	SMC_AXIS_GROUP_INVALID_STATE_INTERNAL_ERROR := 13011,
	SMC_AXIS_GROUP_PCS_INTERNAL_ERROR := 13012,
	SMC_AXIS_GROUP_INTERRUPT_INTERNAL_ERROR := 13013,
	SMC_CONTINUE_DATA_READ_INTERNAL_ERROR := 13014,
	SMC_CONTINUE_DATA_WRITE_INTERNAL_ERROR := 13015,
	SMC_PATH_ELEM_INTERNAL_ERROR := 13016,
	SMC_PATH_ELEM_ESTIMATE_LIMITS_INTERNAL_ERROR := 13017,
	SMC_PATH_ELEM_ZERO_LEN_INTERNAL_ERROR := 13018,
	SMC_PATH_ELEM_BLEND_INTERNAL_ERROR := 13019,
	SMC_PATH_ELEM_BLEND_GEO_INTERNAL_ERROR := 13020,
	SMC_PATH_ELEM_BLEND_ORI_INTERNAL_ERROR := 13021,
	SMC_PATH_ELEM_BLEND_AS_INTERNAL_ERROR := 13022,
	SMC_ELEM_FUN_CART_INTERNAL_ERROR := 13023,
	SMC_CP_HALT_STOP_INTERNAL_ERROR := 13024,
	SMC_TRJ_PLANNING_INIT_INTERNAL_ERROR := 13025,
	SMC_TRJ_PLANNING_GEN_SAMPLES_INTERNAL_ERROR := 13026,
	SMC_TRJ_PLANNING_PATH_OUT_INTERNAL_ERROR := 13027,
	SMC_TRJ_PLANNING_EVAL_AXIS_INTERNAL_ERROR := 13028,
	SMC_TRJ_PLANNING_LOOKAHEAD_INTERNAL_ERROR := 13029,
	SMC_AXIS_GROUP_READ_JERK_INTERNAL_ERROR := 13030,
	SMC_AXIS_GROUP_WRITE_CONTINUE_POS_INTERNAL_ERROR := 13031,
	SMC_CP_TRANSITION_CHECK_FAILED := 13032,
	SMC_ABORTING_INTERNAL_ERROR := 13033,
	SMC_LINE_TO_REL_STANDSTILL_INTERNAL_ERROR := 13034,
	SMC_PATH_ELEM_POSE_EVAL_INTERNAL_ERROR := 13035,
	SMC_CS_REF_COUNT_INTERNAL_ERROR := 13036,
	SMC_PATH_QUEUE_INTERNAL_ERROR := 13037,
	SMC_PATH_ELEM_QUEUE_INTERNAL_ERROR := 13038,
	SMC_ELEM_FUN_QUEUE_INTERNAL_ERROR := 13039,
	SMC_MAC_DUPLICATE_CALLER_INTERNAL_ERROR := 13040,
	SMC_MAC_INTERNAL_ERROR := 13041,
	SMC_READ_POSITION_INTERNAL_ERROR := 13042,
	SMC_ELEM_FUN_PROJECT_POINT_INTERNAL_ERROR := 13043,
	SMC_CAM_EVAL_INTERNAL_ERROR := 13044,
	SMC_CAM_BUILDER_INTERNAL_ERROR_INVALID_CAM_SEGMENT_TYPE := 13045,
	SMC_CAM_BUILDER_INTERNAL_ERROR_INVALID_DESCRIPTION_TYPE := 13046,
	SMC_CAM_BUILDER_INTERNAL_ERROR_IMPLICIT_BOUNDARY_CANNOT_BE_EVALUATED := 13047,
	SMC_CAM_BUILDER_INTERNAL_ERROR_OUT_OF_BOUNDS := 13048,
	SMC_AXIS_MOVEMENTS_INTERNAL_ERROR := 13070,
	SMC_STOP_INTERNAL_ERROR := 13071
) WORD;
END_TYPE

// Device/Application/0.TaskData/TimeManager_Structs/TYPE_
{attribute 'strict'}
TYPE TYPE_ :
(
	TIME_,
    INT_,
    UINT_,
    REAL_
);
END_TYPE

// Device/Application/1.IO/Output/DQ_VARS
{attribute 'strict'}
TYPE DQ_VARS :
(
	outPowerLightColumn	,
	outRedLightColumn 	,
	outGreenLightColumn	,
	outBuzzerLightColumn,
	outExciter			,
	outRemoveLimitSwitch,
	outBit6				,
	outBit7				,
	outBit8				,
	outBit9				,
	outBit10			,
	outBit11			,
	outBit12			,
	outBit13			,
	outBit14			,
	outBit15				
);
END_TYPE

// Device/Application/5.PRG/MAIN
PROGRAM MAIN
VAR
// Блок с данными о времени
	TimeManagerEx	: TimeManager;
// Блок с данными входных сигналов
	InputManagerEx	: InputManager;
// Логика управления стэндом
	StandLogicEx	: StandLogic;
// Блок туправления сервоприводом
	ServoDriverEx	: SM3ServoDriver;
// Блок пегулятора
	PIDControllerEx	: BasicPIDController;
// Блок с данными выходных сигналов
	OutputManagerEx	: OutputManager;
END_VAR

// Данные задачи
TimeManagerEx();

// Входные данные
InputManagerEx();

// Логика управления стэндом
StandLogicEx(
		TimeManager			:= TimeManagerEx,
		InputManager		:= InputManagerEx,
		PIDController		:= PIDControllerEx,
		ServoDriver			:= ServoDriverEx,
 		OutputManager		:= OutputManagerEx);	
			
// Регулятор		
PIDControllerEx();
	
// Сервопривод	
ServoDriverEx(TimeManager := TimeManagerEx);		
		
// Пишем выходные данные		
OutputManagerEx();

END_PROGRAM

// Device/Application/0.TaskData/TimeManager
FUNCTION_BLOCK TimeManager
VAR
	/// Дескриптор (handle) задачи *)
	hTask: CmpIecTask.RTS_IEC_HANDLE;
	/// Результат выполнения функций *)
	result: CmpIecTask.RTS_IEC_RESULT;
	///Указатель на структуру с информацией о задаче *)
	pCurrentTaskInfo: POINTER TO CmpIecTask.Task_Info2;
	///Сама структура с данными *)
	CurrentTaskInfo: CmpIecTask.Task_Info2;
	
	DateAndTime : DTU.GetDateAndTime;
	_dateAndTime : DT;
END_VAR


// 1. Получаем дескриптор текущей задачи
hTask := CmpIecTask.IecTaskGetCurrent(pResult := ADR(result));

// 2. Если дескриптор получен успешно, запрашиваем информацию о задаче
IF hTask <> 0 THEN
    // IecTaskGetInfo3 возвращает указатель на структуру данных о задаче
    pCurrentTaskInfo := CmpIecTask.IecTaskGetInfo3(hIecTask := hTask, pResult := ADR(result));
    
    // 3. Если указатель действителен, копируем данные в нашу локальную переменную
    IF pCurrentTaskInfo <> 0 THEN
        CurrentTaskInfo := pCurrentTaskInfo^;
    END_IF 
END_IF


DateAndTime(xExecute := TRUE);
	IF DateAndTime.xDone THEN
		_dateAndTime := DateAndTime.dtDateAndTime;
		DateAndTime(xExecute := FALSE);
	END_IF

METHOD PUBLIC get_date_time : DT
VAR_INPUT
END_VAR
get_date_time := _dateAndTime;
END_METHOD

METHOD PUBLIC get_interval_time_type_INT : INT;
VAR_INPUT
	measurementUnits	: MEASUREMENT_UNITS;
END_VAR
CASE measurementUnits OF
	MS:                               
		get_interval_time_type_INT  := DWORD_TO_INT(CurrentTaskInfo.dwInterval / 1000);
	US:                                          
		get_interval_time_type_INT := DWORD_TO_INT(CurrentTaskInfo.dwInterval);
END_CASE
END_METHOD

METHOD PUBLIC get_interval_time_type_REAL : REAL;
VAR_INPUT
	measurementUnits	: MEASUREMENT_UNITS;
END_VAR
CASE measurementUnits OF
	MS:                               
		get_interval_time_type_REAL  := DWORD_TO_REAL(CurrentTaskInfo.dwInterval / 1000);
	US:                              
		get_interval_time_type_REAL  := DWORD_TO_REAL(CurrentTaskInfo.dwInterval);
END_CASE
END_METHOD

METHOD PUBLIC get_interval_time_type_TIME : TIME
VAR_INPUT
	measurementUnits	: MEASUREMENT_UNITS;
END_VAR
CASE measurementUnits OF
	MS:                               
		get_interval_time_type_TIME  := DWORD_TO_TIME(CurrentTaskInfo.dwInterval / 1000);
	US:                                          
		get_interval_time_type_TIME  := DWORD_TO_time(CurrentTaskInfo.dwInterval);
END_CASE
END_METHOD

METHOD PUBLIC get_interval_time_type_UINT : UINT;
VAR_INPUT
	measurementUnits	: MEASUREMENT_UNITS;
END_VAR
CASE measurementUnits OF
	MS:                               
		get_interval_time_type_UINT  := DWORD_TO_UINT(CurrentTaskInfo.dwInterval / 1000);
	US:                                          
		get_interval_time_type_UINT  := DWORD_TO_uint(CurrentTaskInfo.dwInterval);
END_CASE
END_METHOD

METHOD PUBLIC get_cycle_count : UDINT
VAR_INPUT
END_VAR
get_cycle_count := DWORD_TO_UDINT(CurrentTaskInfo.dwCycleCount);
END_METHOD

END_FUNCTION_BLOCK

// Device/Application/1.IO/Input/InputManager
FUNCTION_BLOCK InputManager
VAR
    InputBytes (*AT %IB0*) : ARRAY[0..1] OF BYTE;   // Физические входы
    bitsInput          : ARRAY[0..15] OF BOOL;  // Логический массив битов
    iByte              : INT;
    iBit               : INT;
	

	inputReals : ARRAY [tenza1000kgSensor..lastAnalogInIndex - 1] OF REAL;
END_VAR

FOR iByte := 0 TO 1 DO
    FOR iBit := 0 TO 7 DO
        bitsInput[iByte*8 + iBit] := (InputBytes[iByte] AND SHL(BYTE#16#01, iBit)) <> 0;
    END_FOR
END_FOR

METHOD PUBLIC get_analog_data : REAL
VAR_INPUT
	varName		: ALL_AI;
	scaling 	: BOOL;
	inMin		: REAL;
	inMax		: REAL;
	scaleMin	: REAL;
	scaleMax	: REAL;
END_VAR
IF scaling THEN
	IF (inMax - inMin) <> 0 THEN
    	get_analog_data := scaleMin + (inputReals[varName]  - inMin) * (scaleMax - scaleMin) / (inMax - inMin);
	ELSE
    	get_analog_data := inMin; 
	END_IF
ELSE	
	get_analog_data := inputReals[varName];
END_IF
END_METHOD

METHOD PUBLIC get_discrete_data : BOOL
VAR_INPUT
	varName : ALL_DI;
END_VAR
get_discrete_data := bitsInput[varName];
END_METHOD

END_FUNCTION_BLOCK

// Device/Application/1.IO/Output/OutputManager
FUNCTION_BLOCK OutputManager
VAR
    OutputBytes (*AT %QB0*)	: ARRAY[0..1] OF BYTE;
    bitsOutput			: ARRAY[0..15] OF BOOL;
    iByte				: INT;
    iBit				: INT;
    tempByte			: BYTE;
END_VAR

FOR iByte := 0 TO 1 DO
    tempByte := 0;
    FOR iBit := 0 TO 7 DO
        tempByte := tempByte OR (SEL(bitsOutput[iByte*8 + iBit], 0,SHL(BYTE#16#01,iBit)));
    END_FOR
    OutputBytes[iByte] := tempByte;
END_FOR

METHOD PUBLIC set_data : BOOL
VAR_INPUT
	varName : DQ_VARS; 
	enable : BOOL := FALSE;
END_VAR
bitsOutput[varName]:= enable;
set_data := bitsOutput[varName];
END_METHOD

END_FUNCTION_BLOCK

// Device/Application/6.Logic/StandLogic
FUNCTION_BLOCK StandLogic
VAR_INPUT
	{attribute 'symbol' := 'none'}
	TimeManager		: REFERENCE TO TimeManager;
	{attribute 'symbol' := 'none'}
	InputManager	: REFERENCE TO InputManager;
	{attribute 'symbol' := 'none'}
	PIDController	: REFERENCE TO BasicPIDController;
	{attribute 'symbol' := 'none'}
	ServoDriver		: REFERENCE TO SM3ServoDriver;	
	{attribute 'symbol' := 'none'}
	OutputManager	: REFERENCE TO OutputManager;
END_VAR
VAR
	{attribute 'symbol' := 'none'}
	isError					: BOOL := FALSE;
	{attribute 'symbol' := 'none'}
	isStateAxisOperational	: BOOL := FALSE;
	{attribute 'symbol' := 'none'}
	isPowerStatus			: BOOL := FALSE;
	{attribute 'symbol' := 'none'}
	isMoving				: BOOL := FALSE;
	{attribute 'symbol' := 'none'}
	powerInclusionComplited : BOOL := FALSE;
	{attribute 'symbol' := 'none'}
	powerShutdownComplited	: BOOL := FALSE;
	{attribute 'symbol' := 'none'}
	_controlMode				: CONTROL_MODE := MANUAL;
	{attribute 'symbol' := 'none'}
	isExciterEnabled : BOOL := FALSE;
	{attribute 'symbol' := 'none'}
	isInputsReaded : BOOL;
	{attribute 'symbol' := 'none'}
	isForceRemoveLimitSwitchOn : BOOL;
	 
	autoMoveStatus		: AUTO_MOVE_STEPS	:= AWAIT;
	objectStatus		: STATUS			:= NOT_COMMUNICATION;

//Все что 
	// Время вкл/откл возбудителя
	waitExciterOnTime	 : TIME:= T#2S;
	waitExciterOffTime	 : TIME:= T#2S;

		
// Команды
	// Включение силовозбудителя
	cmdExciterOnOff			: BOOL;
	cmdDisableExciter		: BOOL;
	cmdPowerOn				: BOOL;
	cmdPowerOff				: BOOL;
	cmdErrorsReset			: BOOL;
	cmdForwardJogging		: BOOL;
	cmdBackwardJogging		: BOOL;
	cmdChangeControlMode	: BOOL;
	
// Ручное перемещение	
	joggingVelocity		: LREAL;
	joggingAcceleration	: LREAL; 
	joggingDeceleration	: LREAL; 
	joggingJerk			: LREAL;
                    
// Ошибки	
	errorExciterEnableTime	: BOOL;
	errorExciterDisableTime : BOOL;
	
	allErrors : ARRAY [0..15] OF BOOL;
	
	isInitialization	: BOOL := TRUE;
	isInitialized		: BOOL := FALSE;
	
	val : REAL;
	cc : INT;
	
	tenzaSensorDataArr		: ARRAY [0..49] OF REAL;
	displacementSensorArr	: ARRAY [0..49] OF REAL;
	nowSetpoint				: REAL := 600.0;
	
		
	qq : BOOL;
	zz : BOOL;
	
	
	
	ExciterOn				: SwitchingWithFeedbackControl;
	ExciterOff				: SwitchingWithFeedbackControl;
	
	RemovingLimitSwitch : SwitchingWithFeedbackControl;
	
	pidStepKp : REAL;
	pidStepKi : REAL;
	pidStepKd : REAL;	
	algSteps : UINT;
	stepFunction : UINT;
	

// Все нужные DI
	diLiveCircuitsDC		: BOOL;
	diFirstAlarmMushroom	: BOOL;
	diSecondAlarmMushroom	: BOOL;
	diLiveCircuitsAC		: BOOL;
	diUpsDC_OK				: BOOL;
	diUpsBattaryBad			: BOOL;
	diUpsBattaryWork		: BOOL;
	diUpperLimitSwitch		: BOOL;
	diLowerLimitSwitch		: BOOL;
	diRemovingLimitSwitch	: BOOL;
	diExciter				: BOOL;
	diLeftDoor				: BOOL;
	diRightDoor				: BOOL;	
// Для поджига DO
	doForcePowerLightColumn	 : BOOL;	
	doForceRedLightColumn 	 : BOOL;	
	doForceGreenLightColumn	 : BOOL;	
	doForceBuzzerLightColumn : BOOL;	
	doForceExciter			 : BOOL;	
    doForceRemoveLimitSwitch : BOOL;	
// Состояние DO	
	doStatePowerLightColumn	 : BOOL;	
	doStateRedLightColumn 	 : BOOL;	
	doStateGreenLightColumn	 : BOOL;	
	doStateBuzzerLightColumn : BOOL;	
	doStateExciter			 : BOOL;	
	doStateRemoveLimitSwitch : BOOL;	
END_VAR

// Чтение дискретных входов
isInputsReaded			:= _read_inputs();

// Проверка состояния силовозбудителя
isExciterEnabled		:= _check_exciter();

// Проверка состояния снятия с концевиков
isForceRemoveLimitSwitchOn := _check_removing_limit_switch();

// Проверка связи с драйвером
isStateAxisOperational	:= ServoDriver.get_axis_communication();
		
// Проверка наличия питания драйвера
isPowerStatus			:= ServoDriver.get_power_status();

IF NOT isInitialized THEN
	isInitialized := _init(TRUE);
ELSE
	// Включение и отключение дравера
	_driver_power(cmdPowerOn, cmdPowerOff);	
	
	// Режим управления
	CASE read_control_mode OF 
		MANUAL: //Ручное управление
			isMoving := _jogging(
							cmdForward 	 := cmdForwardJogging,
							cmdBackward  := cmdBackwardJogging,
							velocity	 := joggingVelocity,	
			         		acceleration := joggingAcceleration,	
			         		deceleration := joggingDeceleration,
			         		jerk		 := joggingJerk);	
							
		AUTO: // Автоматическое по алгоритму
			;
	END_CASE
	

END_IF
	














 
 IF cc >= 49 THEN
	cc := 0;
ELSE
	cc:= cc + 1;
END_IF

IF val  = 1000 THEN
	qq := TRUE;
	zz := FALSE;
ELSIF val = 0 THEN
	qq := FALSE;
	zz := TRUE;
END_IF

IF qq THEN 
		val := val - 1;
ELSIF zz THEN 
	val := val + 1;
END_IF


tenzaSensorDataArr[cc] := val;
displacementSensorArr[cc] := val + 100.0;
	

	
	//Сброс ошибок
	_reset_alarms(cmdErrorsReset);

	



	

	

	
	
	
	
	
// При аварии колонна подсвечивается красным и включается зуммер
_alarm_notification(FALSE);

// Запись статуса
objectStatus := _get_status();

// Запись выходов
_write_outputs();

METHOD PRIVATE _move_algorythm : BOOL
VAR_INPUT
	enable : BOOL;
	kp : REAL;
	ki : REAL;
	kd : REAL;
	min_out : REAL;
	max_out : REAL;
	pv : REAL;
	sp : REAL;
	laststep : BOOL;
END_VAR
IF enable THEN
	PIDController.Set_Configuration(
								Kp		:= kp,
								Ki		:= ki,
								Kd		:= kd,
								MinOut	:= min_out,
								MaxOut	:= max_out,
								Ts		:= TimeManager.get_interval_time_type_TIME(ms),
	);
															
PIDController.Enable();



PIDController.Reset();

PIDController.Get_Diagnostics();



// Управление скоростью
_move_algorythm := ServoDriver.start_follow_velocity(PIDController.xOutput);

ELSE
	PIDController.Disable();
	_move_algorythm := ServoDriver.stop_follow_velocity();
END_IF
END_METHOD

METHOD PRIVATE _get_status : STATUS
VAR_INPUT
END_VAR
IF isError THEN
    _get_status := ERROR;
ELSIF NOT isStateAxisOperational THEN
    _get_status := NOT_COMMUNICATION;
ELSIF NOT isPowerStatus THEN
    _get_status := OFF;
ELSIF isMoving THEN
    _get_status := MOVING;
ELSE
    _get_status := READY;
END_IF
END_METHOD

METHOD PRIVATE _change_control_mode : CONTROL_MODE
VAR_IN_OUT
	changeMode : BOOL;
END_VAR
IF changeMode THEN
	IF isMoving THEN
		changeMode := FALSE;
	ELSE 
		IF (_controlMode = MANUAL) THEN
			_controlMode := AUTO;
			changeMode	:= FALSE;
		ELSIF (_controlMode = AUTO) THEN
			_controlMode := MANUAL;
			changeMode	:= FALSE;
		END_IF
	END_IF
END_IF

_change_control_mode := _controlMode;
END_METHOD

METHOD PRIVATE _jogging : BOOL
VAR_INPUT
	cmdForward		: BOOL;		// Команда на прямое перемещение
	cmdBackward		: BOOL;		// Команда на обратное перемещение
	velocity		: LREAL;	// Скорость перемещения
	acceleration	: LREAL; 	// Ускорение
	deceleration	: LREAL; 	// Замедление
	jerk			: LREAL;	// Резкость ускорения
END_VAR
END_METHOD

METHOD PRIVATE _init : BOOL
VAR_INPUT
	execute : BOOL;
	exciterEnable	: BOOL := FALSE;
	LimitSwitch		: BOOL := FALSE;
	
END_VAR
VAR
	vv : BYTE;
END_VAR


ServoDriver.set_power_on();
doForceExciter				:= TRUE;
doForceRemoveLimitSwitch	:= FALSE;


vv.0 := exciterEnable;

_init :=  isError;
END_METHOD

//Поджигает светосигнальную колонну красным 
METHOD PRIVATE _alarm_notification : BOOL
VAR_INPUT
	alarm : BOOL := FALSE;
END_VAR
IF alarm THEN 
	OutputManager.set_data(varName := outRedLightColumn,	enable := TRUE);
	OutputManager.set_data(varName := outBuzzerLightColumn, enable := TRUE);
ELSE
	OutputManager.set_data(varName := outRedLightColumn,	enable := FALSE);
	OutputManager.set_data(varName := outBuzzerLightColumn, enable := FALSE);
END_IF
END_METHOD

METHOD PRIVATE _read_inputs : BOOL
VAR_INPUT
END_VAR
diLiveCircuitsDC		:= InputManager.get_discrete_data(inLiveCircuitsDC);
diFirstAlarmMushroom	:= InputManager.get_discrete_data(inFirstAlarmMushroom);
diSecondAlarmMushroom	:= InputManager.get_discrete_data(inSecondAlarmMushroom);
diLiveCircuitsAC		:= InputManager.get_discrete_data(inLiveCircuitsAC);
diUpsDC_OK				:= InputManager.get_discrete_data(inUpsDC_OK);
diUpsBattaryBad			:= InputManager.get_discrete_data(inUpsBattaryBad);
diUpsBattaryWork		:= InputManager.get_discrete_data(inUpsBattaryWork);
diUpperLimitSwitch		:= InputManager.get_discrete_data(inUpperLimitSwitch);
diLowerLimitSwitch		:= InputManager.get_discrete_data(inLowerLimitSwitch);
diRemovingLimitSwitch	:= InputManager.get_discrete_data(inRemovingLimitSwitch);
diExciter				:= InputManager.get_discrete_data(inExciter);
diLeftDoor				:= InputManager.get_discrete_data(inLeftDoor);
diRightDoor				:= InputManager.get_discrete_data(inRightDoor);

_read_inputs := TRUE;
END_METHOD

METHOD PRIVATE _collect_errors : BOOL
VAR_INPUT

END_VAR
VAR	
	i : ERROR_INDEX;
	errors : WORD;
END_VAR


FOR i := communication TO lastIndex - 1 DO
    IF ServoDriver.get_axis_errors(i) THEN
        errors := errors OR SHL(WORD#1, i);
    ELSE
        errors := errors AND NOT SHL(WORD#1, i);
    END_IF
END_FOR

IF errors > 0 THEN
	objectStatus := ERROR;
END_IF
END_METHOD

//Включение и отключение драйвера
METHOD PRIVATE _driver_power : BOOL
VAR_IN_OUT
// Команда на включение
	PowerOnCmd : BOOL; 
// Команда на отключение
	PowerOffCmd : BOOL;
END_VAR
// Входные аргументы методов включения и отключения драйвера
// нужны для корретного завершения вызова методов.
// Т.к логика методов работает по шагам,
// на следующих циклах после начала выполнения метода,
// isPowerStatus сигнализирует о включенном питании,
// тем самым заставляя метод прервать выполнение логики

// Включение
IF PowerOnCmd THEN
	IF powerInclusionComplited := ServoDriver.set_power_on(isPowerStatus AND powerInclusionComplited) THEN
		powerInclusionComplited := FALSE;
		PowerOnCmd				:= FALSE;
	END_IF
	// Отключение
ELSIF PowerOffCmd THEN
	IF powerShutdownComplited := ServoDriver.set_power_off(NOT isPowerStatus AND powerShutdownComplited) THEN 
		powerShutdownComplited	:= FALSE;
		PowerOffCmd				:= FALSE;
	END_IF
END_IF
END_METHOD

METHOD PRIVATE _write_outputs : BOOL
VAR_INPUT
END_VAR
doStatePowerLightColumn		:= OutputManager.set_data(outPowerLightColumn	, doForcePowerLightColumn);	 
doStateRedLightColumn 	 	:= OutputManager.set_data(outRedLightColumn		, doForceRedLightColumn); 	 
doStateGreenLightColumn		:= OutputManager.set_data(outGreenLightColumn	, doForceGreenLightColumn);	 
doStateBuzzerLightColumn	:= OutputManager.set_data(outBuzzerLightColumn	, doForceBuzzerLightColumn);
doStateExciter		   		:= OutputManager.set_data(outExciter			, doForceExciter);		 
doStateRemoveLimitSwitch	:= OutputManager.set_data(outRemoveLimitSwitch	, doForceRemoveLimitSwitch);
END_METHOD

METHOD PRIVATE _reset_alarms : BOOL
VAR_INPUT
	ResetError : BOOL;
END_VAR
IF ResetError THEN 
	IF ServoDriver.reset_errors() THEN 
	;
	END_IF
	cmdErrorsReset := FALSE;
END_IF
END_METHOD

METHOD PRIVATE _check_exciter : BOOL
VAR_INPUT
END_VAR
_check_exciter := diExciter AND doStateExciter;
END_METHOD

{attribute 'monitoring' := 'variable'}
PROPERTY PUBLIC read_control_mode : CONTROL_MODE;
GET

read_control_mode := _controlMode;
END_GET
END_PROPERTY

METHOD PRIVATE _check_removing_limit_switch : BOOL
VAR_INPUT
END_VAR
_check_removing_limit_switch := diRemovingLimitSwitch AND doStateRemoveLimitSwitch;
END_METHOD

END_FUNCTION_BLOCK

// Device/Application/2.PID/BasicPIDController
FUNCTION_BLOCK BasicPIDController

VAR
	_Pv: REAL;
	_Sp: REAL;
	_Kp: REAL;
	_Ki: REAL;
	_Kd: REAL;
	_Ts: TIME;
	_Error: REAL;
	_Output: REAL;
	_MinOut: REAL;
	_MaxOut: REAL;
	_Direction: PID_DIRECTION_UDT;
	_PreviousError: REAL;
	_Proportional: REAL;
	_Integral: REAL;
	_Differential: REAL;
	_Status: PID_STATUS_UDT;
END_VAR

//Включение ПИД
IF _Status <> Enabled THEN
	Reset();	//Integral := 0; PreviousError := 0;Output := 0;
	RETURN;
ELSE
//Значение текущей ошибки
_Error			:= xError(); //CASE Direction OF DIRECT:xError := (Sp - Pv) * 1.0; REVERSE:xError := (Sp - Pv) * -1.0; END_CASE
// Пропорционал
_Proportional	:= xProportional();	//xProportional := Kp * Error;
// Интеграл
_Integral		:= xIntegral();	//xIntegral := LIMIT(OutMin, (Integral + Ki * Error * ((TIME_TO_REAL (Ts)) / 1000)), OutMax);
// ДиФФеренциал
_Differential	:= xDifferential(); //xDifferential := Kd * (Error - PreviousError) / ((TIME_TO_REAL (Ts)) / 1000);
//Значение предыдущей ошибки
_PreviousError	:= _Error;
//Выход ПИД
_Output := LIMIT(_MinOut, _Proportional + _Integral + _Differential, _MaxOut);
END_IF

METHOD Set_Configuration : BOOL
VAR_INPUT
	Kp			: REAL := 0.1;
	Ki			: REAL := 0.0;
	Kd			: REAL := 0;
	Ts			: TIME := T#100MS;
	MinOut		: REAL := 0.0;
	MaxOut		: REAL := 100.0;
	Direction	: PID_DIRECTION_UDT := DIRECT;
END_VAR
_Kp 		 := Kp;		
_Ki 		 := Ki;		
_Kd 		 := Kd;		
_Ts			 := Ts;		
_MinOut		 := MinOut;		
_MaxOut		 := MaxOut;	
_Direction   := Direction;
END_METHOD

METHOD Get_Diagnostics : PID_DIAGNOSTIC_UDT
Get_Diagnostics.Error			:= _Error;			      
Get_Diagnostics.PreviousError	:= _PreviousError;			
Get_Diagnostics.Proportional	:= _Proportional;	 		
Get_Diagnostics.Integral		:= _Integral;		    	
Get_Diagnostics.Differential	:= _Differential;	 		
Get_Diagnostics.Direction		:= _Direction;		   	
Get_Diagnostics.Status			:= _Status;			     
Get_Diagnostics.Kp 				:= _Kp; 		  
Get_Diagnostics.Ki 				:= _Ki; 		  
Get_Diagnostics.Kd 				:= _Kd; 		  
Get_Diagnostics.Ts				:= _Ts;	   
Get_Diagnostics.MinOut			:= _MinOut;	
Get_Diagnostics.MaxOut			:= _MaxOut;
END_METHOD

METHOD PRIVATE xDifferential : REAL
xDifferential := _Kd * (_Error - _PreviousError) / ((TIME_TO_REAL (_Ts)) / 1000);
END_METHOD

METHOD Enable : BOOL
_Status := Enabled;
END_METHOD

METHOD Disable : BOOL
_Status := Disabled;
END_METHOD

PROPERTY xSp : REAL
SET
_Sp := xSp;
END_SET
GET
xSp := _Sp;
END_GET
END_PROPERTY

METHOD PRIVATE xError : REAL
CASE _Direction OF
DIRECT:
	xError := (_Sp - _Pv) * 1.0;
REVERSE:
	xError := (_Sp - _Pv) * -1.0;
END_CASE
END_METHOD

PROPERTY xPv : REAL
GET
xPv := _Pv;
END_GET
SET
_Pv := xPv;
END_SET
END_PROPERTY

METHOD PRIVATE xIntegral : REAL
xIntegral := LIMIT(_MinOut, (_Integral + _Ki * _Error * ((TIME_TO_REAL (_Ts)) / 1000)), _MaxOut);
END_METHOD

PROPERTY xOutput : REAL
SET
END_SET
GET
xOutput := _Output;
END_GET
END_PROPERTY

METHOD Reset : BOOL
_Error			:= 0;
_Integral		:= 0;
_PreviousError	:= 0;
_Output 		:= 0;
END_METHOD

METHOD PRIVATE xProportional : REAL
xProportional := _Kp * _Error;
END_METHOD

END_FUNCTION_BLOCK

// Device/Application/4.Servo/SM3ServoDriver
FUNCTION_BLOCK SM3ServoDriver
VAR_INPUT
	TimeManager		: REFERENCE TO TimeManager;
END_VAR
VAR	
// Проверка  связи с драйвером
	_CheckAxisCommuniction : SMC_CheckAxisCommunication;
//Прверка питания драйвера
	_CheckPowerStatus	: MC_ReadBoolParameter;
	_pNum				: UINT;
	_powerStatusValue	: ARRAY [0..1] OF BOOL;
// Управление питанием драйвера
	_Power		: MC_Power;
	_powerSteps	: UINT;
//Ручной режим
	_Jogging				: MC_Jog;
//Режим управления скоростью
	_FollowVelocity			: SMC_FollowVelocity;
// Сброс аварий
	_Reset_Errors 			: MC_Reset;
	_reset_Enable			: BOOL;
// Дата и время для логов
	
// Сбор ошобок в слово
	_bErrors			: ARRAY [communication..lastIndex - 1] OF BOOL;
	_wAxisErrors		: BYTE;
	_ErrorsFlag			: BOOL;
// 	Данные для флагов ошибок и записи в лог
	_eAxisErrorsID	: ARRAY [communication..lastIndex - 1] OF SMC_ERROR;
	_sComments		: ARRAY [communication..lastIndex - 1] OF STRING(40);
	_trErrorsTrigs	: ARRAY [communication..lastIndex - 1] OF R_TRIG;		
// Лог
	_axisErrorsLog	: ARRAY [0..9] OF STRING(100);
	_logSize		: UINT;
	_errorIndex		: ERROR_INDEX;
END_VAR
VAR CONSTANT
	dPowerParameter: ARRAY [0..1] OF DINT := [1015, 1016];
END_VAR

// Проверка связи
_CheckAxisCommuniction(
	Axis	:= SM_Drive_GenericDSP402,
	bEnable := TRUE);

//Проверка наличия питания
FOR _pNum := 0 TO 1 DO
	_CheckPowerStatus(
		Axis			:= SM_Drive_GenericDSP402,
		Enable			:= TRUE,
		ParameterNumber	:= dPowerParameter[_pNum],
		Value			=> _powerStatusValue[_pNum]); 
END_FOR

// Питание драйвера
_Power(Axis	:= SM_Drive_GenericDSP402);

// Ручное управление дравером
_Jogging(Axis := SM_Drive_GenericDSP402); 

//Режим управления скоростью
_FollowVelocity(Axis := SM_Drive_GenericDSP402);

// Сброс ошибок
_Reset_Errors(Axis:= SM_Drive_GenericDSP402, Execute:= _reset_Enable); 

// // Запись флагов ошибок ФБ в массив
// _bErrors[communication]	 := _CheckAxisCommuniction.bError;
// _bErrors[power]			 := _Power.Error;
// _bErrors[jogging]		 := _Jogging.Error;
// _bErrors[follow]		 := _FollowVelocity.bError;
// _bErrors[reset]			 := _Reset_Errors.Error;

// Запись ошибок
FOR _errorIndex := communication TO lastIndex - 1 DO
	// Триггеры ошибок для записи в лог	
	_trErrorsTrigs[_errorIndex](CLK := _bErrors[_errorIndex]);
	
	// 	Формирование слова ошибок
    IF _bErrors[_errorIndex] THEN
        _wAxisErrors := _wAxisErrors OR SHL(BYTE#1, _errorIndex);
	ELSE
		_wAxisErrors := _wAxisErrors AND NOT SHL(BYTE#1, _errorIndex);
    END_IF
	
END_FOR

// Идентификаторы ошибок
_eAxisErrorsID	[communication]	:= _CheckAxisCommuniction.eErrorID;
_eAxisErrorsID	[power]			:= _Power.ErrorID;
_eAxisErrorsID	[jogging]		:= _Jogging.ErrorID;
_eAxisErrorsID	[follow]		:= _FollowVelocity.iErrorID;
_eAxisErrorsID	[reset]			:= _Reset_Errors.ErrorID;

//Коментарии к ошибкам
_sComments		[communication] := 'Ошибка при диагностике связи';
_sComments		[power]			:= 'Ошибка при включении питания драйвера';
_sComments		[jogging]		:= 'Ошибка при ручном управлении';
_sComments		[follow]		:= 'Ошибка при управлении скоростью';
_sComments		[reset]			:= 'Ошибка при сбросе ошибок';

// Метод для записи ошибки в лог
FOR _errorIndex := communication TO lastIndex - 1 DO
_error_handler(
	bError		:= _trErrorsTrigs[_errorIndex].Q,
	arrIndex	:= _errorIndex,
	eErrorID	:= _eAxisErrorsID[_errorIndex],
	sComment	:= _sComments[_errorIndex]
);	
END_FOR

_ErrorsFlag	:= _wAxisErrors > 0;

METHOD PRIVATE _error_handler : BOOL
VAR_INPUT
	bError   : BOOL;
	arrIndex : ERROR_INDEX;
	eErrorID : SMC_ERROR;
	sComment : STRING;
END_VAR
VAR
	sDT : STRING;
	toStringError : SMC_ERROR_TO_STRING;
END_VAR
// Запускаем блок даты и времени
IF bError THEN
// Приводим дату и время к типу STRING
	sDT := (DT_TO_STRING(TimeManager.get_date_time()));
// Проиводим SMC_ERROR к перечислению которое умеет в TO_STRING
	toStringError := TO_WORD(eErrorID);
// Cобираем сообщение	
	_axisErrorsLog[_logSize] := CONCAT(RIGHT(sDT,LEN(sDT)-3),': ');
	_axisErrorsLog[_logSize] := CONCAT(_axisErrorsLog[_logSize], TO_STRING(toStringError));
	_axisErrorsLog[_logSize] := CONCAT(_axisErrorsLog[_logSize],' ,');
	_axisErrorsLog[_logSize] := CONCAT(_axisErrorsLog[_logSize],sComment);
// Двигаем индекс массива	
	IF _logSize >= 9 THEN
		_logSize := 0;
	ELSE	
		_logSize := _logSize + 1;
	END_IF	
END_IF
END_METHOD

METHOD PUBLIC set_power_on : BOOL
VAR_INPUT
	powerState : BOOL := FALSE;
END_VAR


CASE _powerSteps OF
	0:
		IF powerState THEN
			set_power_on := _Power.Status;
		ELSE
			_powerSteps	:= _powerSteps + 1;	
		END_IF
		
	1: 
		_Power.Enable		:= TRUE;
		_Power.bRegulatorOn := TRUE;
		_Power.bDriveStart	:= TRUE;
		_powerSteps			:= _powerSteps + 1;
	2:
		IF _Power.Status THEN 
			_Power.Enable	:= FALSE;
			_powerSteps		:= _powerSteps + 1;
		END_IF
	3: 
			_Power.bRegulatorOn := FALSE;
			_Power.bDriveStart	:= FALSE;
			set_power_on		:= TRUE;
			_powerSteps			:= 0;
END_CASE
END_METHOD

METHOD PUBLIC stop_follow_velocity : BOOL
VAR_INPUT
END_VAR
_FollowVelocity.bExecute		:= FALSE;
_FollowVelocity.fSetVelocity	:= 0.0; 
	
stop_follow_velocity := _FollowVelocity.bBusy;
END_METHOD

METHOD PUBLIC start_forward_jogging : BOOL
VAR_INPUT
	velocity		: LREAL := 0;
	acceleration	: LREAL := 0;
	deceleration    : LREAL := 0;
	jerk            : LREAL := 0;
END_VAR
_Jogging.JogForward		:= TRUE; 
_Jogging.JogBackward	:= FALSE; 
_Jogging.Velocity		:= velocity; 
_Jogging.Acceleration	:= acceleration; 
_Jogging.Deceleration	:= deceleration; 
_Jogging.Jerk			:= jerk; 

start_forward_jogging := _Jogging.Busy;
END_METHOD

// Проверка питания драйвера
METHOD PUBLIC get_power_status : BOOL
VAR_INPUT
END_VAR
get_power_status := _powerStatusValue[0] AND _powerStatusValue[1] AND _Power.Status AND _Power.Status;
END_METHOD

METHOD PUBLIC set_power_off : BOOL
VAR_INPUT
	powerState : BOOL;
END_VAR
IF powerState THEN
	set_power_off := TRUE;
	RETURN;
ELSE
	CASE _powerSteps OF
		0: 
			_Power.Enable		:= TRUE;
			_Power.bRegulatorOn := FALSE;
			_Power.bDriveStart	:= FALSE;
			_powerSteps			:= _powerSteps + 1;
		1:
			_Power.Enable	:= FALSE;
			_powerSteps			:= _powerSteps + 1;
		2:
			IF NOT _Power.Status THEN
				set_power_off	:= TRUE;
				_powerSteps		:= 0;
			END_IF
	END_CASE
END_IF
END_METHOD

METHOD PUBLIC stop_jogging : BOOL
VAR_INPUT
	velocity		: LREAL := 0;
	acceleration	: LREAL := 0;
	deceleration    : LREAL := 0;
	jerk            : LREAL := 0;
END_VAR
_Jogging.JogForward		:= FALSE; 
_Jogging.JogBackward	:= FALSE; 
_Jogging.Velocity		:= 0; 
_Jogging.Acceleration	:= 0; 
_Jogging.Deceleration	:= 0; 
_Jogging.Jerk			:= 0; 

stop_jogging := _Jogging.Busy;
END_METHOD

METHOD PUBLIC reset_errors : BOOL
VAR_INPUT
END_VAR
_reset_Enable := TRUE;
IF _Reset_Errors.Done THEN
	reset_errors := _Reset_Errors.Done;
	_reset_Enable := FALSE;
END_IF
END_METHOD

METHOD PUBLIC start_follow_velocity : BOOL
VAR_INPUT
	velocity 	: LREAL := 0;
END_VAR
_FollowVelocity.bExecute		:= TRUE;
_FollowVelocity.fSetVelocity	:= velocity; 
	
start_follow_velocity := _FollowVelocity.bBusy;
END_METHOD

METHOD PUBLIC get_axis_errors : BOOL
VAR_INPUT
	errorIndex : ERROR_INDEX;
END_VAR


get_axis_errors := _bErrors[errorIndex];
END_METHOD

METHOD PUBLIC start_backward_jogging : BOOL
VAR_INPUT
	velocity		: LREAL := 0;
	acceleration	: LREAL := 0;
	deceleration    : LREAL := 0;
	jerk            : LREAL := 0;
END_VAR
_Jogging.JogForward		:= FALSE; 
_Jogging.JogBackward	:= TRUE; 
_Jogging.Velocity		:= velocity; 
_Jogging.Acceleration	:= acceleration; 
_Jogging.Deceleration	:= deceleration; 
_Jogging.Jerk			:= jerk; 

start_backward_jogging := _Jogging.Busy;
END_METHOD

//Поверка связи с дравером
METHOD PUBLIC get_axis_communication : BOOL
VAR_INPUT
END_VAR
get_axis_communication := _CheckAxisCommuniction.bOperational;
END_METHOD

END_FUNCTION_BLOCK

// Device/Application/2.Exciter/SwitchingAndFeedbackControl/SwitchingWithFeedbackControl
FUNCTION_BLOCK SwitchingWithFeedbackControl
VAR_INPUT
	xEnable 				: BOOL	:= FALSE;
	xInputSignal			: BOOL	:= FALSE;
	xOutputSignal			: BOOL	:= FALSE;
	waitTimeSwitch			: TIME  := T#2S;
END_VAR
VAR
	WaitingTimer			: WaitingTimer;
END_VAR
VAR_OUTPUT
	xForceOutputSignal		: BOOL:= FALSE;
	xSelfStatus				: SW_STATUS := SW_STATUS.NONE;
END_VAR

// Если нет команды — ничего не делаем
IF NOT xEnable THEN
		WaitingTimer(xExecute := FALSE);
		xForceOutputSignal	:= FALSE;
		xSelfStatus			:= SW_STATUS.NONE;
    RETURN;
END_IF

// Если выход ещё не включён — включаем
IF NOT xOutputSignal THEN
    xForceOutputSignal := TRUE;
    RETURN;
END_IF

// Запуск таймера ожидания обратной связи
WaitingTimer(
    xExecute		:= TRUE,
    xCondition		:= xInputSignal,
    tWaitingTime	:= waitTimeSwitch);
	xSelfStatus := SW_STATUS.WAITING;

// Обратная связь получена
IF WaitingTimer.xDone THEN
    WaitingTimer(xExecute := FALSE);
    xSelfStatus	 := SW_STATUS.DONE;

// Таймаут
ELSIF WaitingTimer.xTimeOutError THEN
    WaitingTimer(xExecute := FALSE);
    xSelfStatus	 := SW_STATUS.TIMEOUT_ERROR;

END_IF

END_FUNCTION_BLOCK

// Device/Application/2.Exciter/SwitchingAndFeedbackControl/WaitingTimer
FUNCTION_BLOCK WaitingTimer
VAR_INPUT
// Включение работы блока
	xExecute		: BOOL := FALSE;
// Ожидаемое состояние
	xCondition		: BOOL := FALSE;
// Максимальное время ожидания состояния
	tWaitingTime	: TIME := T#2S;
END_VAR
VAR_OUTPUT
	//Флаг успешного ожидания состояния
	xDone : BOOL;
	//Флаг ошибки, отсутствие успешного выполнения за заданное время ожидания.
	xTimeOutError : BOOL;
END_VAR
VAR
// Дескриптор (handle) задачи *)
	hTask: CmpIecTask.RTS_IEC_HANDLE;
// Результат выполнения функций *)
	result: CmpIecTask.RTS_IEC_RESULT;
//Указатель на структуру с информацией о задаче *)
	pCurrentTaskInfo: POINTER TO CmpIecTask.Task_Info2;
//Сама структура с данными *)
	CurrentTaskInfo: CmpIecTask.Task_Info2;
// Время цикла в мс
	intervalTime	: TIME;
// Накопленное время
	accumulatedTime : TIME;
END_VAR

// Запись дескриптора текущей задачи в локальную переменную
hTask := CmpIecTask.IecTaskGetCurrent(pResult := ADR(result));

// При успешном получении дискриптора 
IF hTask <> 0 THEN
	// Запрос информации о задаче
    // IecTaskGetInfo3 возвращает указатель на структуру данных о задаче
    pCurrentTaskInfo := CmpIecTask.IecTaskGetInfo3(hIecTask := hTask, pResult := ADR(result));
    // При действительном  указателе, 
    IF pCurrentTaskInfo <> 0 THEN
		// Запись данных в локальную переменную
        CurrentTaskInfo := pCurrentTaskInfo^;
    END_IF 
END_IF

// Записываем полученное время интервала
intervalTime := DWORD_TO_TIME(CurrentTaskInfo.dwInterval / 1000);

//При включении
IF xExecute THEN
	// При отсутвии ошибок
	IF NOT xTimeOutError THEN
		// При наличии требуемого состояния
		IF xCondition AND NOT xTimeOutError THEN 
			// Флаг успешного ожидания
			xDone				:= TRUE;
			// Сброс накопленного времени ожидания
			accumulatedTime		:= T#0MS;
		// При отсутсвии требуемого состояния и отсутствии ошибок
		ELSE
			// Накопление времени ожидания
			accumulatedTime  := accumulatedTime + intervalTime;
			// При достижении максимального времени ожидания
			IF accumulatedTime >= tWaitingTime THEN
				// Флаг ошибки
				xTimeOutError			:= TRUE;
				// Сброс накопленного времени ожидания
				accumulatedTime := T#0MS;
			END_IF
		END_IF
	END_IF
ELSE 
	// Сброс флага успешного ожидания
	xDone				:= FALSE;
	// Сброс флага ошибки
	xTimeOutError		:= FALSE;
	// Сброс накопленного времени ожидания
	accumulatedTime		:= T#0MS;
END_IF

END_FUNCTION_BLOCK

// ГОСТ/Р ИСО 10328-2021/TestingForces_10328
FUNCTION_BLOCK TestingForces_10328
VAR_INPUT
	P : E_P3_8;
	I_II : E_I_II;
END_VAR
VAR_OUTPUT
	Fstab				: UDINT;
	Fset				: UDINT;
	Fsp					: UDINT;
	F_su_lower_level	: UDINT;
	F_su_upper_level	: UDINT;
END_VAR
VAR
END_VAR

CASE P OF
	
	P3:
		CASE I_II OF
			I: 
				Fstab				:= 50;
				Fset				:= 736;
				Fsp					:= 1610;	
 				F_su_lower_level	:= 2415;		
				F_su_upper_level	:= 3220;
			II:   
				Fstab				:= 50;
				Fset				:= 638; 
				Fsp					:= 1395;
				F_su_lower_level	:= 2092;
				F_su_upper_level	:= 2790;
		END_CASE
		
	P4:
		CASE I_II OF
			I: 
				Fstab				:= 50;
				Fset				:= 944; 
				Fsp					:= 2065;
				F_su_lower_level	:= 3098;
				F_su_upper_level	:= 4130;
			II: 
				Fstab				:= 50;
				Fset				:= 828; 
				Fsp					:= 1811; 
				F_su_lower_level	:= 2717;
				F_su_upper_level	:= 3623;
		END_CASE
		
	P5:
		CASE I_II OF
			I: 
				Fstab				:= 50;
				Fset				:= 1024;
				Fsp					:= 2240;
				F_su_lower_level	:= 3360;
				F_su_upper_level	:= 4480;
			II:  
				Fstab 				:= 50; 
				Fset  				:= 920;
				Fsp					:= 2013;	
				F_su_lower_level	:= 3019;
				F_su_upper_level	:= 4025;
		END_CASE	
		
	P6:
		CASE I_II OF
			I: 
				Fstab				:= 50;
				Fset				:= 1224;
				Fsp					:= 2490;
				F_su_lower_level	:= 3760;
				F_su_upper_level	:= 4480;
			II:  
				Fstab 				:= 50; 
				Fset  				:= 1120;
				Fsp					:= 2263;	
				F_su_lower_level	:= 3419;
				F_su_upper_level	:= 4425;
		END_CASE	
		
	P7:
		CASE I_II OF
			I: 
				Fstab				:= 50;
				Fset				:= 1416;
				Fsp					:= 2900;
				F_su_lower_level	:= 4100;
				F_su_upper_level	:= 5300;
			II:  
				Fstab 				:= 50; 
				Fset  				:= 1360;
				Fsp					:= 2650;	
				F_su_lower_level	:= 3775;
				F_su_upper_level	:= 4840;
		END_CASE		
		
	P8:
		CASE I_II OF
			I: 
				Fstab				:= 50;
				Fset				:= 1640;
				Fsp					:= 3200;
				F_su_lower_level	:= 4450;
				F_su_upper_level	:= 5700;
			II:  
				Fstab 				:= 50; 
				Fset  				:= 1560;
				Fsp					:= 2950;	
				F_su_lower_level	:= 4150;
				F_su_upper_level	:= 5250;
		END_CASE	
END_CASE

END_FUNCTION_BLOCK

// ГОСТ/ Р53868-2021/TestingForces_53868
FUNCTION_BLOCK TestingForces_53868
VAR_INPUT
	P : E_P1_2;
	I_II : E_I_II;
END_VAR
VAR_OUTPUT
	Fstab				: UDINT;
	Fset				: UDINT;
	Fsp					: UDINT;
	F_su_lower_level	: UDINT;
	F_su_upper_level	: UDINT;
END_VAR
VAR
END_VAR

CASE P OF
	
	P1:
		CASE I_II OF
			I: 
				Fstab				:= 50;
// 				Fset				:= 736;
// 				Fsp					:= 1610;	
 				F_su_lower_level	:= 930;		
				F_su_upper_level	:= 1240;
			II:   
				Fstab				:= 50;
// 				Fset				:= 638; 
// 				Fsp					:= 1395;
				F_su_lower_level	:= 825;
				F_su_upper_level	:= 1100;
		END_CASE
		
	P2:
		CASE I_II OF
			I: 
				Fstab				:= 50;
// 				Fset				:= 944; 
// 				Fsp					:= 2065;
				F_su_lower_level	:= 1680;
				F_su_upper_level	:= 2250;
			II: 
				Fstab				:= 50;
// 				Fset				:= 828; 
// 				Fsp					:= 1811; 
				F_su_lower_level	:= 1490;
				F_su_upper_level	:= 1990;
		END_CASE
END_CASE

END_FUNCTION_BLOCK

// ГОСТ/Р ИСО 15032-2001/TestingForces_150321
FUNCTION_BLOCK TestingForces_150321
VAR_INPUT
	A : E_A;
END_VAR
VAR_OUTPUT
	Fstab				: UDINT;
	Fset				: UDINT;
	Fsp					: UDINT;
	F_su_lower_level	: UDINT;
	F_su_upper_level	: UDINT;
END_VAR
VAR
END_VAR

CASE A OF
	
	A60:
				Fstab				:= 50;
				Fset				:= 720;
				Fsp					:= 1575;	
				
 				F_su_lower_level	:= 2363;		
				F_su_upper_level	:= 3150;
	
	A80: 
				Fstab				:= 50;
				Fset				:= 840; 
				Fsp					:= 1838;
				
				F_su_lower_level	:= 2756;
				F_su_upper_level	:= 3675;

	A100:
				Fstab				:= 50;
				Fset				:= 1024;
				Fsp					:= 2240;
				
				F_su_lower_level	:= 3360;
				F_su_upper_level	:= 4480;
						
END_CASE

END_FUNCTION_BLOCK
